LIN {X 0,Y 400.277,Z 579.545,A -85,B 0,C 180,E1 -11266.71,E2 -11266.71} C_VEL
LIN {X 0,Y 401.436,Z 567.994,A -85,B 0,C 180,E1 -11267.974,E2 -11267.974} C_VEL
LIN {X 0,Y 402.651,Z 555.178,A -85,B 0,C 180,E1 -11269.104,E2 -11269.104} C_VEL
LIN {X 0,Y 403.742,Z 541.629,A -85,B 0,C 180,E1 -11270.046,E2 -11270.046} C_VEL
LIN {X 0,Y 404.528,Z 528.73,A -85,B 0,C 180,E1 -11270.732,E2 -11270.732} C_VEL
LIN {X 0,Y 405.302,Z 514.967,A -85,B 0,C 180,E1 -11271.256,E2 -11271.256} C_VEL
LIN {X 0,Y 405.728,Z 500.889,A -85,B 0,C 180,E1 -11271.599,E2 -11271.599} C_VEL
LIN {X 0,Y 407.367,Z 401.658,A -85,B 0,C 180,E1 -11273.361,E2 -11273.361} C_VEL
LIN {X 0,Y 404.27,Z 384.321,A -85,B 0,C 180,E1 -11273.88,E2 -11273.88} C_VEL
LIN {X 0,Y 401.419,Z 370.358,A -85,B 0,C 180,E1 -11274.356,E2 -11274.356} C_VEL
LIN {X 0,Y 401.756,Z 366.638,A -85,B 0,C 180,E1 -11275.102,E2 -11275.102} C_VEL
LIN {X 0,Y 399.711,Z 355.979,A -85,B 0,C 180,E1 -11277.471,E2 -11277.471} C_VEL
LIN {X 0,Y 397.114,Z 344.644,A -85,B 0,C 180,E1 -11280.118,E2 -11280.118} C_VEL
LIN {X 0,Y 397.123,Z 344.645,A -85,B 0,C 180,E1 -11283.719,E2 -11283.719} C_VEL
LIN {X 0,Y 397.098,Z 344.645,A -85,B 0,C 180,E1 -11287.21,E2 -11287.21} C_VEL
LIN {X 0,Y 397.107,Z 344.641,A -85,B 0,C 180,E1 -11290.446,E2 -11290.446} C_VEL
LIN {X 0,Y 397.106,Z 344.644,A -85,B 0,C 180,E1 -11293.649,E2 -11293.649} C_VEL
LIN {X 0,Y 397.107,Z 344.643,A -85,B 0,C 180,E1 -11296.522,E2 -11296.522} C_VEL
LIN {X 0,Y 397.119,Z 344.642,A -85,B 0,C 180,E1 -11300.423,E2 -11300.423} C_VEL
LIN {X 0,Y 397.113,Z 344.646,A -85,B 0,C 180,E1 -11304.266,E2 -11304.266} C_VEL
LIN {X 0,Y 397.12,Z 344.644,A -85,B 0,C 180,E1 -11306.728,E2 -11306.728} C_VEL
LIN {X 0,Y 397.124,Z 344.649,A -85,B 0,C 180,E1 -11310.296,E2 -11310.296} C_VEL
LIN {X 0,Y 397.16,Z 344.763,A -85,B 0,C 180,E1 -11311.134,E2 -11311.134} C_VEL
LIN {X 0,Y 400.789,Z 356.95,A -85,B 0,C 180,E1 -11313.999,E2 -11313.999} C_VEL
LIN {X 0,Y 402.495,Z 364.53,A -85,B 0,C 180,E1 -11315.662,E2 -11315.662} C_VEL
LIN {X 0,Y 402.859,Z 369.281,A -85,B 0,C 180,E1 -11316.617,E2 -11316.617} C_VEL
LIN {X 0,Y 402.299,Z 381.598,A -85,B 0,C 180,E1 -11318.881,E2 -11318.881} C_VEL
LIN {X 0,Y 405.879,Z 396.627,A -85,B 0,C 180,E1 -11319.635,E2 -11319.635} C_VEL
LIN {X 0,Y 406.448,Z 400.682,A -85,B 0,C 180,E1 -11319.801,E2 -11319.801} C_VEL
LIN {X 0,Y 403.617,Z 480.645,A -85,B 0,C 180,E1 -11321.8,E2 -11321.8} C_VEL
LIN {X 0,Y 403.108,Z 495.536,A -85,B 0,C 180,E1 -11322.236,E2 -11322.236} C_VEL
LIN {X 0,Y 402.537,Z 508.176,A -85,B 0,C 180,E1 -11322.8,E2 -11322.8} C_VEL
LIN {X 0,Y 401.908,Z 519.55,A -85,B 0,C 180,E1 -11323.492,E2 -11323.492} C_VEL
LIN {X 0,Y 401.064,Z 531.353,A -85,B 0,C 180,E1 -11324.409,E2 -11324.409} C_VEL
LIN {X 0,Y 400.264,Z 541.681,A -85,B 0,C 180,E1 -11325.417,E2 -11325.417} C_VEL
LIN {X 0,Y 399.455,Z 550.912,A -85,B 0,C 180,E1 -11326.519,E2 -11326.519} C_VEL
LIN {X 0,Y 398.69,Z 559.636,A -85,B 0,C 180,E1 -11327.788,E2 -11327.788} C_VEL
LIN {X 0,Y 397.891,Z 568.178,A -85,B 0,C 180,E1 -11329.312,E2 -11329.312} C_VEL
LIN {X 0,Y 397.225,Z 574.98,A -85,B 0,C 180,E1 -11330.838,E2 -11330.838} C_VEL
LIN {X 0,Y 396.781,Z 580.383,A -85,B 0,C 180,E1 -11332.367,E2 -11332.367} C_VEL
LIN {X 0,Y 396.415,Z 584.568,A -85,B 0,C 180,E1 -11333.894,E2 -11333.894} C_VEL
LIN {X 0,Y 396.15,Z 586.768,A -85,B 0,C 180,E1 -11334.911,E2 -11334.911} C_VEL
LIN {X 0,Y 396.205,Z 588.437,A -85,B 0,C 180,E1 -11335.931,E2 -11335.931} C_VEL
LIN {X 0,Y 396.084,Z 589.693,A -85,B 0,C 180,E1 -11336.949,E2 -11336.949} C_VEL
LIN {X 0,Y 395.941,Z 590.539,A -85,B 0,C 180,E1 -11337.966,E2 -11337.966} C_VEL
LIN {X 0,Y 395.859,Z 590.913,A -85,B 0,C 180,E1 -11338.983,E2 -11338.983} C_VEL
LIN {X 0,Y 395.823,Z 590.865,A -85,B 0,C 180,E1 -11340,E2 -11340} C_VEL
LIN {X 0,Y 395.838,Z 590.407,A -85,B 0,C 180,E1 -11341.017,E2 -11341.017} C_VEL
LIN {X 0,Y 395.919,Z 589.489,A -85,B 0,C 180,E1 -11342.035,E2 -11342.035} C_VEL
LIN {X 0,Y 395.951,Z 588.135,A -85,B 0,C 180,E1 -11343.052,E2 -11343.052} C_VEL
LIN {X 0,Y 395.996,Z 585.27,A -85,B 0,C 180,E1 -11344.581,E2 -11344.581} C_VEL
LIN {X 0,Y 396.189,Z 581.317,A -85,B 0,C 180,E1 -11346.11,E2 -11346.11} C_VEL
LIN {X 0,Y 396.423,Z 576.171,A -85,B 0,C 180,E1 -11347.641,E2 -11347.641} C_VEL
LIN {X 0,Y 396.767,Z 569.656,A -85,B 0,C 180,E1 -11349.173,E2 -11349.173} C_VEL
LIN {X 0,Y 397.271,Z 561.487,A -85,B 0,C 180,E1 -11350.705,E2 -11350.705} C_VEL
LIN {X 0,Y 397.764,Z 553.153,A -85,B 0,C 180,E1 -11351.982,E2 -11351.982} C_VEL
LIN {X 0,Y 398.467,Z 542.953,A -85,B 0,C 180,E1 -11353.255,E2 -11353.255} C_VEL
LIN {X 0,Y 399.008,Z 532.049,A -85,B 0,C 180,E1 -11354.358,E2 -11354.358} C_VEL
LIN {X 0,Y 399.571,Z 520.38,A -85,B 0,C 180,E1 -11355.298,E2 -11355.298} C_VEL
LIN {X 0,Y 400.209,Z 506.876,A -85,B 0,C 180,E1 -11356.122,E2 -11356.122} C_VEL
LIN {X 0,Y 400.642,Z 493.868,A -85,B 0,C 180,E1 -11356.693,E2 -11356.693} C_VEL
LIN {X 0,Y 400.978,Z 479.075,A -85,B 0,C 180,E1 -11357.105,E2 -11357.105} C_VEL
LIN {X 0,Y 402.535,Z 397.502,A -85,B 0,C 180,E1 -11358.899,E2 -11358.899} C_VEL
LIN {X 0,Y 399.311,Z 377.922,A -85,B 0,C 180,E1 -11359.487,E2 -11359.487} C_VEL
LIN {X 0,Y 399.99,Z 360.43,A -85,B 0,C 180,E1 -11362.74,E2 -11362.74} C_VEL
LIN {X 0,Y 398.852,Z 353.072,A -85,B 0,C 180,E1 -11364.185,E2 -11364.185} C_VEL
LIN {X 0,Y 397.174,Z 344.638,A -85,B 0,C 180,E1 -11365.907,E2 -11365.907} C_VEL
LIN {X 0,Y 397.128,Z 344.643,A -85,B 0,C 180,E1 -11368.543,E2 -11368.543} C_VEL
LIN {X 0,Y 397.085,Z 344.649,A -85,B 0,C 180,E1 -11372.071,E2 -11372.071} C_VEL
LIN {X 0,Y 397.125,Z 344.642,A -85,B 0,C 180,E1 -11375.503,E2 -11375.503} C_VEL
LIN {X 0,Y 397.099,Z 344.643,A -85,B 0,C 180,E1 -11378.854,E2 -11378.854} C_VEL
LIN {X 0,Y 397.067,Z 344.65,A -85,B 0,C 180,E1 -11382.268,E2 -11382.268} C_VEL
LIN {X 0,Y 397.092,Z 344.646,A -85,B 0,C 180,E1 -11385.068,E2 -11385.068} C_VEL
LIN {X 0,Y 397.059,Z 344.651,A -85,B 0,C 180,E1 -11388.023,E2 -11388.023} C_VEL
LIN {X 0,Y 397.095,Z 344.648,A -85,B 0,C 180,E1 -11391.723,E2 -11391.723} C_VEL
LIN {X 0,Y 397.122,Z 344.641,A -85,B 0,C 180,E1 -11395.505,E2 -11395.505} C_VEL
LIN {X 0,Y 397.076,Z 344.649,A -85,B 0,C 180,E1 -11399.116,E2 -11399.116} C_VEL
LIN {X 0,Y 397.131,Z 344.765,A -85,B 0,C 180,E1 -11401.203,E2 -11401.203} C_VEL
LIN {X 0,Y 399.898,Z 357.338,A -85,B 0,C 180,E1 -11404.215,E2 -11404.215} C_VEL
LIN {X 0,Y 401.222,Z 363.882,A -85,B 0,C 180,E1 -11405.714,E2 -11405.714} C_VEL
LIN {X 0,Y 403.242,Z 371.317,A -85,B 0,C 180,E1 -11405.986,E2 -11405.986} C_VEL
LIN {X 0,Y 407.408,Z 391.656,A -85,B 0,C 180,E1 -11406.631,E2 -11406.631} C_VEL
LIN {X 0,Y 405.903,Z 489.536,A -85,B 0,C 180,E1 -11408.377,E2 -11408.377} C_VEL
LIN {X 0,Y 405.462,Z 505.277,A -85,B 0,C 180,E1 -11408.719,E2 -11408.719} C_VEL
LIN {X 0,Y 404.756,Z 519.212,A -85,B 0,C 180,E1 -11409.213,E2 -11409.213} C_VEL
LIN {X 0,Y 404.017,Z 532.788,A -85,B 0,C 180,E1 -11409.906,E2 -11409.906} C_VEL
LIN {X 0,Y 403.024,Z 545.847,A -85,B 0,C 180,E1 -11410.782,E2 -11410.782} C_VEL
LIN {X 0,Y 401.966,Z 557.736,A -85,B 0,C 180,E1 -11411.787,E2 -11411.787} C_VEL
LIN {X 0,Y 400.713,Z 569.777,A -85,B 0,C 180,E1 -11413.046,E2 -11413.046} C_VEL
LIN {X 0,Y 399.899,Z 577.879,A -85,B 0,C 180,E1 -11414.06,E2 -11414.06} C_VEL
LIN {X 0,Y 398.895,Z 580.792,A -85,B 0,C 180,E1 -11414.427,E2 -11414.427} C_VEL
LIN {X 0,Y 392.324,Z 589.579,A -85,B 0,C 180,E1 -11415.574,E2 -11415.574} C_VEL
LIN {X 0,Y 391.485,Z 592.107,A -85,B 0,C 180,E1 -11416.004,E2 -11416.004} C_VEL
LIN {X 0,Y 390.581,Z 600.976,A -85,B 0,C 180,E1 -11417.793,E2 -11417.793} C_VEL
LIN {X 0,Y 389.828,Z 608.252,A -85,B 0,C 180,E1 -11419.612,E2 -11419.612} C_VEL
LIN {X 0,Y 389.212,Z 614.788,A -85,B 0,C 180,E1 -11421.693,E2 -11421.693} C_VEL
LIN {X 0,Y 388.924,Z 619.682,A -85,B 0,C 180,E1 -11423.774,E2 -11423.774} C_VEL
LIN {X 0,Y 388.718,Z 623.093,A -85,B 0,C 180,E1 -11425.851,E2 -11425.851} C_VEL
LIN {X 0,Y 388.66,Z 625.122,A -85,B 0,C 180,E1 -11427.926,E2 -11427.926} C_VEL
LIN {X 0,Y 388.672,Z 625.82,A -85,B 0,C 180,E1 -11429.998,E2 -11429.998} C_VEL
LIN {X 0,Y 388.659,Z 625.196,A -85,B 0,C 180,E1 -11432.071,E2 -11432.071} C_VEL
LIN {X 0,Y 388.716,Z 623.237,A -85,B 0,C 180,E1 -11434.146,E2 -11434.146} C_VEL
LIN {X 0,Y 388.873,Z 619.891,A -85,B 0,C 180,E1 -11436.224,E2 -11436.224} C_VEL
LIN {X 0,Y 389.207,Z 615.06,A -85,B 0,C 180,E1 -11438.304,E2 -11438.304} C_VEL
LIN {X 0,Y 389.799,Z 608.599,A -85,B 0,C 180,E1 -11440.385,E2 -11440.385} C_VEL
LIN {X 0,Y 390.544,Z 601.405,A -85,B 0,C 180,E1 -11442.205,E2 -11442.205} C_VEL
LIN {X 0,Y 391.402,Z 592.717,A -85,B 0,C 180,E1 -11443.987,E2 -11443.987} C_VEL
LIN {X 0,Y 392.456,Z 583.155,A -85,B 0,C 180,E1 -11445.58,E2 -11445.58} C_VEL
LIN {X 0,Y 393.642,Z 572.796,A -85,B 0,C 180,E1 -11446.997,E2 -11446.997} C_VEL
LIN {X 0,Y 394.857,Z 561.37,A -85,B 0,C 180,E1 -11448.281,E2 -11448.281} C_VEL
LIN {X 0,Y 396.091,Z 548.705,A -85,B 0,C 180,E1 -11449.43,E2 -11449.43} C_VEL
LIN {X 0,Y 397.149,Z 535.171,A -85,B 0,C 180,E1 -11450.402,E2 -11450.402} C_VEL
LIN {X 0,Y 398.085,Z 521.413,A -85,B 0,C 180,E1 -11451.148,E2 -11451.148} C_VEL
LIN {X 0,Y 398.801,Z 507.58,A -85,B 0,C 180,E1 -11451.685,E2 -11451.685} C_VEL
LIN {X 0,Y 399.296,Z 493.25,A -85,B 0,C 180,E1 -11452.03,E2 -11452.03} C_VEL
LIN {X 0,Y 400.989,Z 393.489,A -85,B 0,C 180,E1 -11453.832,E2 -11453.832} C_VEL
LIN {X 0,Y 396.082,Z 369.523,A -85,B 0,C 180,E1 -11454.614,E2 -11454.614} C_VEL
LIN {X 0,Y 394.027,Z 363.86,A -85,B 0,C 180,E1 -11454.87,E2 -11454.87} C_VEL
LIN {X 0,Y 391.431,Z 351.504,A -85,B 0,C 180,E1 -11457.826,E2 -11457.826} C_VEL
LIN {X 0,Y 390.083,Z 345.525,A -85,B 0,C 180,E1 -11459.327,E2 -11459.327} C_VEL
LIN {X 0,Y 390.036,Z 345.531,A -85,B 0,C 180,E1 -11462.72,E2 -11462.72} C_VEL
LIN {X 0,Y 390.048,Z 345.525,A -85,B 0,C 180,E1 -11465.823,E2 -11465.823} C_VEL
LIN {X 0,Y 390.029,Z 345.527,A -85,B 0,C 180,E1 -11469.211,E2 -11469.211} C_VEL
LIN {X 0,Y 390.021,Z 345.527,A -85,B 0,C 180,E1 -11472.37,E2 -11472.37} C_VEL
LIN {X 0,Y 390.033,Z 345.525,A -85,B 0,C 180,E1 -11475.352,E2 -11475.352} C_VEL
LIN {X 0,Y 390.005,Z 345.528,A -85,B 0,C 180,E1 -11478.183,E2 -11478.183} C_VEL
LIN {X 0,Y 390.047,Z 345.519,A -85,B 0,C 180,E1 -11480.902,E2 -11480.902} C_VEL
LIN {X 0,Y 390.07,Z 345.524,A -85,B 0,C 180,E1 -11484.791,E2 -11484.791} C_VEL
LIN {X 0,Y 390.009,Z 345.52,A -85,B 0,C 180,E1 -11488.494,E2 -11488.494} C_VEL
LIN {X 0,Y 390.002,Z 345.524,A -85,B 0,C 180,E1 -11492.002,E2 -11492.002} C_VEL
LIN {X 0,Y 390.029,Z 345.522,A -85,B 0,C 180,E1 -11495.516,E2 -11495.516} C_VEL
LIN {X 0,Y 390.041,Z 345.517,A -85,B 0,C 180,E1 -11498.877,E2 -11498.877} C_VEL
LIN {X 0,Y 390.097,Z 345.504,A -85,B 0,C 180,E1 -11502.165,E2 -11502.165} C_VEL
LIN {X 0,Y 390.126,Z 345.511,A -85,B 0,C 180,E1 -11505.392,E2 -11505.392} C_VEL
LIN {X 0,Y 390.13,Z 345.515,A -85,B 0,C 180,E1 -11508.571,E2 -11508.571} C_VEL
LIN {X 0,Y 390.241,Z 345.495,A -85,B 0,C 180,E1 -11512.086,E2 -11512.086} C_VEL
LIN {X 0,Y 390.184,Z 345.502,A -85,B 0,C 180,E1 -11514.833,E2 -11514.833} C_VEL
LIN {X 0,Y 390.395,Z 345.479,A -85,B 0,C 180,E1 -11517.937,E2 -11517.937} C_VEL
LIN {X 0,Y 390.392,Z 345.48,A -85,B 0,C 180,E1 -11522.063,E2 -11522.063} C_VEL
LIN {X 0,Y 390.269,Z 345.496,A -85,B 0,C 180,E1 -11526.203,E2 -11526.203} C_VEL
LIN {X 0,Y 390.17,Z 345.504,A -85,B 0,C 180,E1 -11529.33,E2 -11529.33} C_VEL
LIN {X 0,Y 390.18,Z 345.502,A -85,B 0,C 180,E1 -11533.439,E2 -11533.439} C_VEL
LIN {X 0,Y 390.115,Z 345.51,A -85,B 0,C 180,E1 -11537.299,E2 -11537.299} C_VEL
LIN {X 0,Y 390.074,Z 345.514,A -85,B 0,C 180,E1 -11540.471,E2 -11540.471} C_VEL
LIN {X 0,Y 390.043,Z 345.513,A -85,B 0,C 180,E1 -11543.354,E2 -11543.354} C_VEL
LIN {X 0,Y 390.018,Z 345.524,A -85,B 0,C 180,E1 -11546.775,E2 -11546.775} C_VEL
LIN {X 0,Y 390.023,Z 345.52,A -85,B 0,C 180,E1 -11550.301,E2 -11550.301} C_VEL
LIN {X 0,Y 390.056,Z 345.521,A -85,B 0,C 180,E1 -11554.026,E2 -11554.026} C_VEL
LIN {X 0,Y 390.023,Z 345.527,A -85,B 0,C 180,E1 -11557.782,E2 -11557.782} C_VEL
LIN {X 0,Y 390.004,Z 345.527,A -85,B 0,C 180,E1 -11560.816,E2 -11560.816} C_VEL
LIN {X 0,Y 390.032,Z 345.525,A -85,B 0,C 180,E1 -11563.886,E2 -11563.886} C_VEL
LIN {X 0,Y 390.036,Z 345.527,A -85,B 0,C 180,E1 -11566.789,E2 -11566.789} C_VEL
LIN {X 0,Y 390,Z 345.531,A -85,B 0,C 180,E1 -11569.556,E2 -11569.556} C_VEL
LIN {X 0,Y 390.027,Z 345.53,A -85,B 0,C 180,E1 -11572.452,E2 -11572.452} C_VEL
LIN {X 0,Y 390.054,Z 345.526,A -85,B 0,C 180,E1 -11576.046,E2 -11576.046} C_VEL
LIN {X 0,Y 390.071,Z 345.654,A -85,B 0,C 180,E1 -11579.518,E2 -11579.518} C_VEL
LIN {X 0,Y 393.033,Z 358.498,A -85,B 0,C 180,E1 -11582.566,E2 -11582.566} C_VEL
LIN {X 0,Y 394.863,Z 367.974,A -85,B 0,C 180,E1 -11584.714,E2 -11584.714} C_VEL
LIN {X 0,Y 394.674,Z 370.357,A -85,B 0,C 180,E1 -11585.203,E2 -11585.203} C_VEL
LIN {X 0,Y 400.422,Z 399.362,A -85,B 0,C 180,E1 -11586.156,E2 -11586.156} C_VEL
LIN {X 0,Y 400.86,Z 403.279,A -85,B 0,C 180,E1 -11586.259,E2 -11586.259} C_VEL
LIN {X 0,Y 399.023,Z 507.416,A -85,B 0,C 180,E1 -11588.158,E2 -11588.158} C_VEL
LIN {X 0,Y 398.362,Z 521.51,A -85,B 0,C 180,E1 -11588.596,E2 -11588.596} C_VEL
LIN {X 0,Y 397.48,Z 535.196,A -85,B 0,C 180,E1 -11589.225,E2 -11589.225} C_VEL
LIN {X 0,Y 396.474,Z 548.971,A -85,B 0,C 180,E1 -11590.087,E2 -11590.087} C_VEL
LIN {X 0,Y 395.362,Z 561.288,A -85,B 0,C 180,E1 -11591.072,E2 -11591.072} C_VEL
LIN {X 0,Y 394.149,Z 572.919,A -85,B 0,C 180,E1 -11592.222,E2 -11592.222} C_VEL
LIN {X 0,Y 393.09,Z 582.602,A -85,B 0,C 180,E1 -11593.379,E2 -11593.379} C_VEL
LIN {X 0,Y 391.871,Z 593.332,A -85,B 0,C 180,E1 -11594.929,E2 -11594.929} C_VEL
LIN {X 0,Y 390.958,Z 602.191,A -85,B 0,C 180,E1 -11596.487,E2 -11596.487} C_VEL
LIN {X 0,Y 390.267,Z 609.564,A -85,B 0,C 180,E1 -11598.05,E2 -11598.05} C_VEL
LIN {X 0,Y 389.589,Z 615.708,A -85,B 0,C 180,E1 -11599.609,E2 -11599.609} C_VEL
LIN {X 0,Y 389.09,Z 622.234,A -85,B 0,C 180,E1 -11601.693,E2 -11601.693} C_VEL
LIN {X 0,Y 388.802,Z 627.209,A -85,B 0,C 180,E1 -11603.817,E2 -11603.817} C_VEL
LIN {X 0,Y 388.681,Z 630.52,A -85,B 0,C 180,E1 -11605.854,E2 -11605.854} C_VEL
LIN {X 0,Y 388.613,Z 632.525,A -85,B 0,C 180,E1 -11607.929,E2 -11607.929} C_VEL
LIN {X 0,Y 388.671,Z 633.187,A -85,B 0,C 180,E1 -11610.002,E2 -11610.002} C_VEL
LIN {X 0,Y 388.614,Z 632.516,A -85,B 0,C 180,E1 -11612.074,E2 -11612.074} C_VEL
LIN {X 0,Y 388.681,Z 630.502,A -85,B 0,C 180,E1 -11614.149,E2 -11614.149} C_VEL
LIN {X 0,Y 388.835,Z 627.099,A -85,B 0,C 180,E1 -11616.227,E2 -11616.227} C_VEL
LIN {X 0,Y 389.093,Z 622.207,A -85,B 0,C 180,E1 -11618.31,E2 -11618.31} C_VEL
LIN {X 0,Y 389.593,Z 615.67,A -85,B 0,C 180,E1 -11620.394,E2 -11620.394} C_VEL
LIN {X 0,Y 390.367,Z 608.398,A -85,B 0,C 180,E1 -11622.214,E2 -11622.214} C_VEL
LIN {X 0,Y 391.12,Z 600.545,A -85,B 0,C 180,E1 -11623.82,E2 -11623.82} C_VEL
LIN {X 0,Y 392.048,Z 591.631,A -85,B 0,C 180,E1 -11625.334,E2 -11625.334} C_VEL
LIN {X 0,Y 393.342,Z 580.542,A -85,B 0,C 180,E1 -11626.88,E2 -11626.88} C_VEL
LIN {X 0,Y 394.533,Z 569.216,A -85,B 0,C 180,E1 -11628.165,E2 -11628.165} C_VEL
LIN {X 0,Y 395.779,Z 556.688,A -85,B 0,C 180,E1 -11629.315,E2 -11629.315} C_VEL
LIN {X 0,Y 396.912,Z 543.713,A -85,B 0,C 180,E1 -11630.259,E2 -11630.259} C_VEL
LIN {X 0,Y 397.796,Z 529.957,A -85,B 0,C 180,E1 -11631.032,E2 -11631.032} C_VEL
LIN {X 0,Y 398.651,Z 515.806,A -85,B 0,C 180,E1 -11631.595,E2 -11631.595} C_VEL
LIN {X 0,Y 399.113,Z 502.36,A -85,B 0,C 180,E1 -11631.942,E2 -11631.942} C_VEL
LIN {X 0,Y 400.848,Z 404.818,A -85,B 0,C 180,E1 -11633.702,E2 -11633.702} C_VEL
LIN {X 0,Y 400.532,Z 399.888,A -85,B 0,C 180,E1 -11633.817,E2 -11633.817} C_VEL
LIN {X 0,Y 394.671,Z 370.347,A -85,B 0,C 180,E1 -11634.788,E2 -11634.788} C_VEL
LIN {X 0,Y 394.677,Z 366.564,A -85,B 0,C 180,E1 -11635.584,E2 -11635.584} C_VEL
LIN {X 0,Y 391.99,Z 353.714,A -85,B 0,C 180,E1 -11638.535,E2 -11638.535} C_VEL
LIN {X 0,Y 390.058,Z 345.525,A -85,B 0,C 180,E1 -11640.524,E2 -11640.524} C_VEL
LIN {X 0,Y 390.073,Z 345.521,A -85,B 0,C 180,E1 -11644.026,E2 -11644.026} C_VEL
LIN {X 0,Y 390.047,Z 345.524,A -85,B 0,C 180,E1 -11647.551,E2 -11647.551} C_VEL
LIN {X 0,Y 390.061,Z 345.52,A -85,B 0,C 180,E1 -11650.822,E2 -11650.822} C_VEL
LIN {X 0,Y 390.06,Z 345.522,A -85,B 0,C 180,E1 -11653.887,E2 -11653.887} C_VEL
LIN {X 0,Y 390.062,Z 345.522,A -85,B 0,C 180,E1 -11656.79,E2 -11656.79} C_VEL
LIN {X 0,Y 390.062,Z 345.521,A -85,B 0,C 180,E1 -11659.561,E2 -11659.561} C_VEL
LIN {X 0,Y 390.048,Z 345.524,A -85,B 0,C 180,E1 -11662.45,E2 -11662.45} C_VEL
LIN {X 0,Y 390.074,Z 345.524,A -85,B 0,C 180,E1 -11666.046,E2 -11666.046} C_VEL
LIN {X 0,Y 390.05,Z 345.53,A -85,B 0,C 180,E1 -11669.87,E2 -11669.87} C_VEL
LIN {X 0,Y 390.08,Z 345.542,A -85,B 0,C 180,E1 -11670.3,E2 -11670.3} C_VEL
LIN {X 0,Y 393.751,Z 357.145,A -85,B 0,C 180,E1 -11673.184,E2 -11673.184} C_VEL
LIN {X 0,Y 395.963,Z 366.556,A -85,B 0,C 180,E1 -11675.32,E2 -11675.32} C_VEL
LIN {X 0,Y 396.421,Z 370.831,A -85,B 0,C 180,E1 -11676.214,E2 -11676.214} C_VEL
LIN {X 0,Y 395.855,Z 382.001,A -85,B 0,C 180,E1 -11678.311,E2 -11678.311} C_VEL
LIN {X 0,Y 399.364,Z 396.308,A -85,B 0,C 180,E1 -11679.08,E2 -11679.08} C_VEL
LIN {X 0,Y 400.252,Z 401.562,A -85,B 0,C 180,E1 -11679.32,E2 -11679.32} C_VEL
LIN {X 0,Y 397.189,Z 480.415,A -85,B 0,C 180,E1 -11681.361,E2 -11681.361} C_VEL
LIN {X 0,Y 396.65,Z 495.328,A -85,B 0,C 180,E1 -11681.803,E2 -11681.803} C_VEL
LIN {X 0,Y 396.046,Z 508.049,A -85,B 0,C 180,E1 -11682.375,E2 -11682.375} C_VEL
LIN {X 0,Y 395.342,Z 519.518,A -85,B 0,C 180,E1 -11683.076,E2 -11683.076} C_VEL
LIN {X 0,Y 394.463,Z 531.491,A -85,B 0,C 180,E1 -11684.022,E2 -11684.022} C_VEL
LIN {X 0,Y 393.51,Z 542.814,A -85,B 0,C 180,E1 -11685.154,E2 -11685.154} C_VEL
LIN {X 0,Y 392.392,Z 553.857,A -85,B 0,C 180,E1 -11686.536,E2 -11686.536} C_VEL
LIN {X 0,Y 391.644,Z 562.12,A -85,B 0,C 180,E1 -11687.828,E2 -11687.828} C_VEL
LIN {X 0,Y 390.865,Z 570.195,A -85,B 0,C 180,E1 -11689.38,E2 -11689.38} C_VEL
LIN {X 0,Y 390.263,Z 575.699,A -85,B 0,C 180,E1 -11690.673,E2 -11690.673} C_VEL
LIN {X 0,Y 389.78,Z 581.03,A -85,B 0,C 180,E1 -11692.228,E2 -11692.228} C_VEL
LIN {X 0,Y 389.387,Z 585.154,A -85,B 0,C 180,E1 -11693.783,E2 -11693.783} C_VEL
LIN {X 0,Y 389.094,Z 587.299,A -85,B 0,C 180,E1 -11694.818,E2 -11694.818} C_VEL
LIN {X 0,Y 389.135,Z 588.926,A -85,B 0,C 180,E1 -11695.857,E2 -11695.857} C_VEL
LIN {X 0,Y 389.03,Z 590.148,A -85,B 0,C 180,E1 -11696.893,E2 -11696.893} C_VEL
LIN {X 0,Y 388.878,Z 590.946,A -85,B 0,C 180,E1 -11697.929,E2 -11697.929} C_VEL
LIN {X 0,Y 388.788,Z 591.276,A -85,B 0,C 180,E1 -11698.964,E2 -11698.964} C_VEL
LIN {X 0,Y 388.75,Z 591.192,A -85,B 0,C 180,E1 -11700,E2 -11700} C_VEL
LIN {X 0,Y 388.768,Z 590.69,A -85,B 0,C 180,E1 -11701.036,E2 -11701.036} C_VEL
LIN {X 0,Y 388.835,Z 589.714,A -85,B 0,C 180,E1 -11702.072,E2 -11702.072} C_VEL
LIN {X 0,Y 388.854,Z 588.322,A -85,B 0,C 180,E1 -11703.108,E2 -11703.108} C_VEL
LIN {X 0,Y 388.931,Z 585.378,A -85,B 0,C 180,E1 -11704.664,E2 -11704.664} C_VEL
LIN {X 0,Y 389.118,Z 581.341,A -85,B 0,C 180,E1 -11706.221,E2 -11706.221} C_VEL
LIN {X 0,Y 389.358,Z 576.096,A -85,B 0,C 180,E1 -11707.781,E2 -11707.781} C_VEL
LIN {X 0,Y 389.736,Z 569.434,A -85,B 0,C 180,E1 -11709.34,E2 -11709.34} C_VEL
LIN {X 0,Y 390.235,Z 561.133,A -85,B 0,C 180,E1 -11710.9,E2 -11710.9} C_VEL
LIN {X 0,Y 390.789,Z 552.648,A -85,B 0,C 180,E1 -11712.199,E2 -11712.199} C_VEL
LIN {X 0,Y 391.452,Z 542.201,A -85,B 0,C 180,E1 -11713.497,E2 -11713.497} C_VEL
LIN {X 0,Y 392.089,Z 530.527,A -85,B 0,C 180,E1 -11714.666,E2 -11714.666} C_VEL
LIN {X 0,Y 392.662,Z 518.966,A -85,B 0,C 180,E1 -11715.574,E2 -11715.574} C_VEL
LIN {X 0,Y 393.289,Z 506.215,A -85,B 0,C 180,E1 -11716.347,E2 -11716.347} C_VEL
LIN {X 0,Y 393.719,Z 492.724,A -85,B 0,C 180,E1 -11716.929,E2 -11716.929} C_VEL
LIN {X 0,Y 394.04,Z 478.712,A -85,B 0,C 180,E1 -11717.316,E2 -11717.316} C_VEL
LIN {X 0,Y 395.663,Z 398.492,A -85,B 0,C 180,E1 -11719.133,E2 -11719.133} C_VEL
LIN {X 0,Y 392.379,Z 378.146,A -85,B 0,C 180,E1 -11719.759,E2 -11719.759} C_VEL
LIN {X 0,Y 393.039,Z 361.462,A -85,B 0,C 180,E1 -11722.887,E2 -11722.887} C_VEL
LIN {X 0,Y 391.522,Z 352.494,A -85,B 0,C 180,E1 -11724.667,E2 -11724.667} C_VEL
LIN {X 0,Y 390.141,Z 345.515,A -85,B 0,C 180,E1 -11726.084,E2 -11726.084} C_VEL
LIN {X 0,Y 390.064,Z 345.52,A -85,B 0,C 180,E1 -11729.109,E2 -11729.109} C_VEL
LIN {X 0,Y 390.049,Z 345.522,A -85,B 0,C 180,E1 -11732.721,E2 -11732.721} C_VEL
LIN {X 0,Y 390.061,Z 345.524,A -85,B 0,C 180,E1 -11735.825,E2 -11735.825} C_VEL
LIN {X 0,Y 390.043,Z 345.522,A -85,B 0,C 180,E1 -11739.212,E2 -11739.212} C_VEL
LIN {X 0,Y 390.042,Z 345.524,A -85,B 0,C 180,E1 -11742.373,E2 -11742.373} C_VEL
LIN {X 0,Y 390.049,Z 345.525,A -85,B 0,C 180,E1 -11745.353,E2 -11745.353} C_VEL
LIN {X 0,Y 390.022,Z 345.527,A -85,B 0,C 180,E1 -11748.184,E2 -11748.184} C_VEL
LIN {X 0,Y 390.062,Z 345.522,A -85,B 0,C 180,E1 -11750.903,E2 -11750.903} C_VEL
LIN {X 0,Y 390.074,Z 345.519,A -85,B 0,C 180,E1 -11754.791,E2 -11754.791} C_VEL
LIN {X 0,Y 390.022,Z 345.529,A -85,B 0,C 180,E1 -11758.494,E2 -11758.494} C_VEL
LIN {X 0,Y 390.091,Z 345.629,A -85,B 0,C 180,E1 -11760.818,E2 -11760.818} C_VEL
LIN {X 0,Y 393.019,Z 358.821,A -85,B 0,C 180,E1 -11764.045,E2 -11764.045} C_VEL
LIN {X 0,Y 394.088,Z 364.135,A -85,B 0,C 180,E1 -11765.248,E2 -11765.248} C_VEL
LIN {X 0,Y 396.357,Z 370.651,A -85,B 0,C 180,E1 -11765.527,E2 -11765.527} C_VEL
LIN {X 0,Y 400.941,Z 393.402,A -85,B 0,C 180,E1 -11766.263,E2 -11766.263} C_VEL
LIN {X 0,Y 399.139,Z 497.863,A -85,B 0,C 180,E1 -11768.162,E2 -11768.162} C_VEL
LIN {X 0,Y 398.592,Z 512.141,A -85,B 0,C 180,E1 -11768.572,E2 -11768.572} C_VEL
LIN {X 0,Y 397.864,Z 524.655,A -85,B 0,C 180,E1 -11769.107,E2 -11769.107} C_VEL
LIN {X 0,Y 396.904,Z 538.586,A -85,B 0,C 180,E1 -11769.917,E2 -11769.917} C_VEL
LIN {X 0,Y 395.874,Z 550.66,A -85,B 0,C 180,E1 -11770.825,E2 -11770.825} C_VEL
LIN {X 0,Y 394.715,Z 562.953,A -85,B 0,C 180,E1 -11771.978,E2 -11771.978} C_VEL
LIN {X 0,Y 393.576,Z 573.051,A -85,B 0,C 180,E1 -11773.13,E2 -11773.13} C_VEL
LIN {X 0,Y 392.489,Z 582.475,A -85,B 0,C 180,E1 -11774.418,E2 -11774.418} C_VEL
LIN {X 0,Y 391.485,Z 592.107,A -85,B 0,C 180,E1 -11776.004,E2 -11776.004} C_VEL
LIN {X 0,Y 390.592,Z 595.757,A -85,B 0,C 180,E1 -11776.675,E2 -11776.675} C_VEL
LIN {X 0,Y 387.181,Z 601.366,A -85,B 0,C 180,E1 -11777.769,E2 -11777.769} C_VEL
LIN {X 0,Y 383.695,Z 606.461,A -85,B 0,C 180,E1 -11778.928,E2 -11778.928} C_VEL
LIN {X 0,Y 382.704,Z 609.251,A -85,B 0,C 180,E1 -11779.692,E2 -11779.692} C_VEL
LIN {X 0,Y 382.159,Z 614.857,A -85,B 0,C 180,E1 -11781.538,E2 -11781.538} C_VEL
LIN {X 0,Y 381.85,Z 619.751,A -85,B 0,C 180,E1 -11783.658,E2 -11783.658} C_VEL
LIN {X 0,Y 381.647,Z 623.16,A -85,B 0,C 180,E1 -11785.774,E2 -11785.774} C_VEL
LIN {X 0,Y 381.558,Z 625.189,A -85,B 0,C 180,E1 -11787.887,E2 -11787.887} C_VEL
LIN {X 0,Y 381.572,Z 625.887,A -85,B 0,C 180,E1 -11789.998,E2 -11789.998} C_VEL
LIN {X 0,Y 381.557,Z 625.263,A -85,B 0,C 180,E1 -11792.11,E2 -11792.11} C_VEL
LIN {X 0,Y 381.645,Z 623.303,A -85,B 0,C 180,E1 -11794.223,E2 -11794.223} C_VEL
LIN {X 0,Y 381.807,Z 619.957,A -85,B 0,C 180,E1 -11796.339,E2 -11796.339} C_VEL
LIN {X 0,Y 382.153,Z 615.126,A -85,B 0,C 180,E1 -11798.459,E2 -11798.459} C_VEL
LIN {X 0,Y 382.773,Z 608.665,A -85,B 0,C 180,E1 -11800.578,E2 -11800.578} C_VEL
LIN {X 0,Y 383.58,Z 601.471,A -85,B 0,C 180,E1 -11802.43,E2 -11802.43} C_VEL
LIN {X 0,Y 384.416,Z 593.319,A -85,B 0,C 180,E1 -11804.139,E2 -11804.139} C_VEL
LIN {X 0,Y 385.399,Z 584.875,A -85,B 0,C 180,E1 -11805.601,E2 -11805.601} C_VEL
LIN {X 0,Y 386.712,Z 573.904,A -85,B 0,C 180,E1 -11807.175,E2 -11807.175} C_VEL
LIN {X 0,Y 387.982,Z 562.72,A -85,B 0,C 180,E1 -11808.48,E2 -11808.48} C_VEL
LIN {X 0,Y 389.255,Z 550.346,A -85,B 0,C 180,E1 -11809.648,E2 -11809.648} C_VEL
LIN {X 0,Y 390.306,Z 537.716,A -85,B 0,C 180,E1 -11810.603,E2 -11810.603} C_VEL
LIN {X 0,Y 391.306,Z 524.07,A -85,B 0,C 180,E1 -11811.395,E2 -11811.395} C_VEL
LIN {X 0,Y 392.109,Z 509.468,A -85,B 0,C 180,E1 -11812.005,E2 -11812.005} C_VEL
LIN {X 0,Y 392.704,Z 494.938,A -85,B 0,C 180,E1 -11812.385,E2 -11812.385} C_VEL
LIN {X 0,Y 394.491,Z 394.763,A -85,B 0,C 180,E1 -11814.226,E2 -11814.226} C_VEL
LIN {X 0,Y 390.195,Z 373.29,A -85,B 0,C 180,E1 -11814.937,E2 -11814.937} C_VEL
LIN {X 0,Y 388.077,Z 367.022,A -85,B 0,C 180,E1 -11815.208,E2 -11815.208} C_VEL
LIN {X 0,Y 386.824,Z 363.961,A -85,B 0,C 180,E1 -11815.358,E2 -11815.358} C_VEL
LIN {X 0,Y 384.222,Z 351.572,A -85,B 0,C 180,E1 -11818.395,E2 -11818.395} C_VEL
LIN {X 0,Y 383.015,Z 346.405,A -85,B 0,C 180,E1 -11819.755,E2 -11819.755} C_VEL
LIN {X 0,Y 382.997,Z 346.406,A -85,B 0,C 180,E1 -11823.399,E2 -11823.399} C_VEL
LIN {X 0,Y 383.024,Z 346.4,A -85,B 0,C 180,E1 -11826.162,E2 -11826.162} C_VEL
LIN {X 0,Y 382.966,Z 346.405,A -85,B 0,C 180,E1 -11829.961,E2 -11829.961} C_VEL
LIN {X 0,Y 382.997,Z 346.402,A -85,B 0,C 180,E1 -11832.777,E2 -11832.777} C_VEL
LIN {X 0,Y 382.985,Z 346.401,A -85,B 0,C 180,E1 -11835.787,E2 -11835.787} C_VEL
LIN {X 0,Y 382.951,Z 346.408,A -85,B 0,C 180,E1 -11838.799,E2 -11838.799} C_VEL
LIN {X 0,Y 382.982,Z 346.393,A -85,B 0,C 180,E1 -11842.096,E2 -11842.096} C_VEL
LIN {X 0,Y 383.005,Z 346.398,A -85,B 0,C 180,E1 -11845.331,E2 -11845.331} C_VEL
LIN {X 0,Y 382.969,Z 346.405,A -85,B 0,C 180,E1 -11849.08,E2 -11849.08} C_VEL
LIN {X 0,Y 382.957,Z 346.394,A -85,B 0,C 180,E1 -11852.69,E2 -11852.69} C_VEL
LIN {X 0,Y 382.996,Z 346.399,A -85,B 0,C 180,E1 -11856.19,E2 -11856.19} C_VEL
LIN {X 0,Y 383.042,Z 346.383,A -85,B 0,C 180,E1 -11859.598,E2 -11859.598} C_VEL
LIN {X 0,Y 383.08,Z 346.387,A -85,B 0,C 180,E1 -11862.93,E2 -11862.93} C_VEL
LIN {X 0,Y 383.112,Z 346.386,A -85,B 0,C 180,E1 -11866.463,E2 -11866.463} C_VEL
LIN {X 0,Y 383.127,Z 346.384,A -85,B 0,C 180,E1 -11870.497,E2 -11870.497} C_VEL
LIN {X 0,Y 383.214,Z 346.372,A -85,B 0,C 180,E1 -11873.682,E2 -11873.682} C_VEL
LIN {X 0,Y 383.361,Z 346.355,A -85,B 0,C 180,E1 -11877.899,E2 -11877.899} C_VEL
LIN {X 0,Y 383.358,Z 346.356,A -85,B 0,C 180,E1 -11882.101,E2 -11882.101} C_VEL
LIN {X 0,Y 383.225,Z 346.375,A -85,B 0,C 180,E1 -11886.317,E2 -11886.317} C_VEL
LIN {X 0,Y 383.121,Z 346.382,A -85,B 0,C 180,E1 -11889.503,E2 -11889.503} C_VEL
LIN {X 0,Y 383.111,Z 346.382,A -85,B 0,C 180,E1 -11893.536,E2 -11893.536} C_VEL
LIN {X 0,Y 383.08,Z 346.387,A -85,B 0,C 180,E1 -11897.07,E2 -11897.07} C_VEL
LIN {X 0,Y 383.015,Z 346.391,A -85,B 0,C 180,E1 -11900.647,E2 -11900.647} C_VEL
LIN {X 0,Y 382.994,Z 346.392,A -85,B 0,C 180,E1 -11903.81,E2 -11903.81} C_VEL
LIN {X 0,Y 382.957,Z 346.401,A -85,B 0,C 180,E1 -11907.31,E2 -11907.31} C_VEL
LIN {X 0,Y 382.968,Z 346.405,A -85,B 0,C 180,E1 -11910.92,E2 -11910.92} C_VEL
LIN {X 0,Y 382.998,Z 346.402,A -85,B 0,C 180,E1 -11914.67,E2 -11914.67} C_VEL
LIN {X 0,Y 382.979,Z 346.405,A -85,B 0,C 180,E1 -11917.903,E2 -11917.903} C_VEL
LIN {X 0,Y 382.948,Z 346.405,A -85,B 0,C 180,E1 -11921.352,E2 -11921.352} C_VEL
LIN {X 0,Y 382.978,Z 346.408,A -85,B 0,C 180,E1 -11924.303,E2 -11924.303} C_VEL
LIN {X 0,Y 382.972,Z 346.405,A -85,B 0,C 180,E1 -11927.238,E2 -11927.238} C_VEL
LIN {X 0,Y 382.974,Z 346.409,A -85,B 0,C 180,E1 -11930.421,E2 -11930.421} C_VEL
LIN {X 0,Y 383.004,Z 346.405,A -85,B 0,C 180,E1 -11934.045,E2 -11934.045} C_VEL
LIN {X 0,Y 382.977,Z 346.406,A -85,B 0,C 180,E1 -11937.58,E2 -11937.58} C_VEL
LIN {X 0,Y 383.007,Z 346.428,A -85,B 0,C 180,E1 -11939.086,E2 -11939.086} C_VEL
LIN {X 0,Y 386.126,Z 359.868,A -85,B 0,C 180,E1 -11942.349,E2 -11942.349} C_VEL
LIN {X 0,Y 387.969,Z 369.226,A -85,B 0,C 180,E1 -11944.516,E2 -11944.516} C_VEL
LIN {X 0,Y 387.918,Z 370.33,A -85,B 0,C 180,E1 -11944.75,E2 -11944.75} C_VEL
LIN {X 0,Y 393.841,Z 399.763,A -85,B 0,C 180,E1 -11945.741,E2 -11945.741} C_VEL
LIN {X 0,Y 394.377,Z 403.386,A -85,B 0,C 180,E1 -11945.847,E2 -11945.847} C_VEL
LIN {X 0,Y 392.453,Z 507.364,A -85,B 0,C 180,E1 -11947.773,E2 -11947.773} C_VEL
LIN {X 0,Y 391.771,Z 521.451,A -85,B 0,C 180,E1 -11948.218,E2 -11948.218} C_VEL
LIN {X 0,Y 390.866,Z 535.135,A -85,B 0,C 180,E1 -11948.857,E2 -11948.857} C_VEL
LIN {X 0,Y 389.831,Z 548.385,A -85,B 0,C 180,E1 -11949.692,E2 -11949.692} C_VEL
LIN {X 0,Y 388.645,Z 561.225,A -85,B 0,C 180,E1 -11950.732,E2 -11950.732} C_VEL
LIN {X 0,Y 387.352,Z 572.854,A -85,B 0,C 180,E1 -11951.9,E2 -11951.9} C_VEL
LIN {X 0,Y 386.252,Z 582.537,A -85,B 0,C 180,E1 -11953.076,E2 -11953.076} C_VEL
LIN {X 0,Y 384.984,Z 593.266,A -85,B 0,C 180,E1 -11954.653,E2 -11954.653} C_VEL
LIN {X 0,Y 384.017,Z 602.125,A -85,B 0,C 180,E1 -11956.238,E2 -11956.238} C_VEL
LIN {X 0,Y 383.273,Z 609.498,A -85,B 0,C 180,E1 -11957.828,E2 -11957.828} C_VEL
LIN {X 0,Y 382.553,Z 615.641,A -85,B 0,C 180,E1 -11959.416,E2 -11959.416} C_VEL
LIN {X 0,Y 382.157,Z 620.731,A -85,B 0,C 180,E1 -11961.008,E2 -11961.008} C_VEL
LIN {X 0,Y 381.78,Z 625.989,A -85,B 0,C 180,E1 -11963.129,E2 -11963.129} C_VEL
LIN {X 0,Y 381.648,Z 628.934,A -85,B 0,C 180,E1 -11964.719,E2 -11964.719} C_VEL
LIN {X 0,Y 381.509,Z 631.625,A -85,B 0,C 180,E1 -11966.834,E2 -11966.834} C_VEL
LIN {X 0,Y 381.551,Z 632.955,A -85,B 0,C 180,E1 -11968.946,E2 -11968.946} C_VEL
LIN {X 0,Y 381.551,Z 632.951,A -85,B 0,C 180,E1 -11971.057,E2 -11971.057} C_VEL
LIN {X 0,Y 381.51,Z 631.61,A -85,B 0,C 180,E1 -11973.17,E2 -11973.17} C_VEL
LIN {X 0,Y 381.648,Z 628.911,A -85,B 0,C 180,E1 -11975.284,E2 -11975.284} C_VEL
LIN {X 0,Y 381.793,Z 625.964,A -85,B 0,C 180,E1 -11976.873,E2 -11976.873} C_VEL
LIN {X 0,Y 382.16,Z 620.7,A -85,B 0,C 180,E1 -11978.995,E2 -11978.995} C_VEL
LIN {X 0,Y 382.557,Z 615.601,A -85,B 0,C 180,E1 -11980.587,E2 -11980.587} C_VEL
LIN {X 0,Y 383.406,Z 608.329,A -85,B 0,C 180,E1 -11982.439,E2 -11982.439} C_VEL
LIN {X 0,Y 384.233,Z 599.81,A -85,B 0,C 180,E1 -11984.205,E2 -11984.205} C_VEL
LIN {X 0,Y 385.387,Z 589.867,A -85,B 0,C 180,E1 -11985.877,E2 -11985.877} C_VEL
LIN {X 0,Y 386.612,Z 579.404,A -85,B 0,C 180,E1 -11987.319,E2 -11987.319} C_VEL
LIN {X 0,Y 387.919,Z 567.852,A -85,B 0,C 180,E1 -11988.623,E2 -11988.623} C_VEL
LIN {X 0,Y 389.252,Z 555.034,A -85,B 0,C 180,E1 -11989.789,E2 -11989.789} C_VEL
LIN {X 0,Y 390.33,Z 542.261,A -85,B 0,C 180,E1 -11990.712,E2 -11990.712} C_VEL
LIN {X 0,Y 391.271,Z 528.582,A -85,B 0,C 180,E1 -11991.469,E2 -11991.469} C_VEL
LIN {X 0,Y 392.11,Z 514.813,A -85,B 0,C 180,E1 -11992.008,E2 -11992.008} C_VEL
LIN {X 0,Y 392.581,Z 500.715,A -85,B 0,C 180,E1 -11992.361,E2 -11992.361} C_VEL
LIN {X 0,Y 394.342,Z 404.73,A -85,B 0,C 180,E1 -11994.118,E2 -11994.118} C_VEL
LIN {X 0,Y 393.952,Z 400.502,A -85,B 0,C 180,E1 -11994.226,E2 -11994.226} C_VEL
LIN {X 0,Y 388.165,Z 371.649,A -85,B 0,C 180,E1 -11995.185,E2 -11995.185} C_VEL
LIN {X 0,Y 387.93,Z 370.259,A -85,B 0,C 180,E1 -11995.253,E2 -11995.253} C_VEL
LIN {X 0,Y 387.198,Z 365.148,A -85,B 0,C 180,E1 -11996.405,E2 -11996.405} C_VEL
LIN {X 0,Y 384.566,Z 352.745,A -85,B 0,C 180,E1 -11999.338,E2 -11999.338} C_VEL
LIN {X 0,Y 383.007,Z 346.402,A -85,B 0,C 180,E1 -12000.918,E2 -12000.918} C_VEL
LIN {X 0,Y 383.023,Z 346.397,A -85,B 0,C 180,E1 -12004.669,E2 -12004.669} C_VEL
LIN {X 0,Y 383.003,Z 346.399,A -85,B 0,C 180,E1 -12007.904,E2 -12007.904} C_VEL
LIN {X 0,Y 382.989,Z 346.404,A -85,B 0,C 180,E1 -12011.348,E2 -12011.348} C_VEL
LIN {X 0,Y 383.001,Z 346.399,A -85,B 0,C 180,E1 -12014.304,E2 -12014.304} C_VEL
LIN {X 0,Y 383.016,Z 346.401,A -85,B 0,C 180,E1 -12017.241,E2 -12017.241} C_VEL
LIN {X 0,Y 383.021,Z 346.398,A -85,B 0,C 180,E1 -12020.414,E2 -12020.414} C_VEL
LIN {X 0,Y 383.03,Z 346.398,A -85,B 0,C 180,E1 -12024.045,E2 -12024.045} C_VEL
LIN {X 0,Y 382.992,Z 346.406,A -85,B 0,C 180,E1 -12027.579,E2 -12027.579} C_VEL
LIN {X 0,Y 383.004,Z 346.446,A -85,B 0,C 180,E1 -12029.389,E2 -12029.389} C_VEL
LIN {X 0,Y 385.986,Z 355.283,A -85,B 0,C 180,E1 -12031.744,E2 -12031.744} C_VEL
LIN {X 0,Y 388.587,Z 364.49,A -85,B 0,C 180,E1 -12034,E2 -12034} C_VEL
LIN {X 0,Y 389.857,Z 371.111,A -85,B 0,C 180,E1 -12035.504,E2 -12035.504} C_VEL
LIN {X 0,Y 389.813,Z 376.763,A -85,B 0,C 180,E1 -12036.632,E2 -12036.632} C_VEL
LIN {X 0,Y 389.539,Z 382.504,A -85,B 0,C 180,E1 -12037.706,E2 -12037.706} C_VEL
LIN {X 0,Y 392.943,Z 396.152,A -85,B 0,C 180,E1 -12038.496,E2 -12038.496} C_VEL
LIN {X 0,Y 394.128,Z 403.129,A -85,B 0,C 180,E1 -12038.832,E2 -12038.832} C_VEL
LIN {X 0,Y 390.835,Z 480.687,A -85,B 0,C 180,E1 -12040.91,E2 -12040.91} C_VEL
LIN {X 0,Y 390.236,Z 495.467,A -85,B 0,C 180,E1 -12041.357,E2 -12041.357} C_VEL
LIN {X 0,Y 389.527,Z 509.354,A -85,B 0,C 180,E1 -12042.003,E2 -12042.003} C_VEL
LIN {X 0,Y 388.743,Z 521.417,A -85,B 0,C 180,E1 -12042.78,E2 -12042.78} C_VEL
LIN {X 0,Y 387.772,Z 533.083,A -85,B 0,C 180,E1 -12043.739,E2 -12043.739} C_VEL
LIN {X 0,Y 386.775,Z 543.953,A -85,B 0,C 180,E1 -12044.87,E2 -12044.87} C_VEL
LIN {X 0,Y 385.576,Z 554.963,A -85,B 0,C 180,E1 -12046.293,E2 -12046.293} C_VEL
LIN {X 0,Y 384.622,Z 564.527,A -85,B 0,C 180,E1 -12047.87,E2 -12047.87} C_VEL
LIN {X 0,Y 383.848,Z 572.224,A -85,B 0,C 180,E1 -12049.45,E2 -12049.45} C_VEL
LIN {X 0,Y 383.093,Z 578.352,A -85,B 0,C 180,E1 -12051.029,E2 -12051.029} C_VEL
LIN {X 0,Y 382.642,Z 583.34,A -85,B 0,C 180,E1 -12052.674,E2 -12052.674} C_VEL
LIN {X 0,Y 382.176,Z 586.849,A -85,B 0,C 180,E1 -12054.195,E2 -12054.195} C_VEL
LIN {X 0,Y 382.069,Z 589.429,A -85,B 0,C 180,E1 -12055.781,E2 -12055.781} C_VEL
LIN {X 0,Y 381.977,Z 590.618,A -85,B 0,C 180,E1 -12056.836,E2 -12056.836} C_VEL
LIN {X 0,Y 381.817,Z 591.349,A -85,B 0,C 180,E1 -12057.89,E2 -12057.89} C_VEL
LIN {X 0,Y 381.72,Z 591.639,A -85,B 0,C 180,E1 -12058.945,E2 -12058.945} C_VEL
LIN {X 0,Y 381.68,Z 591.519,A -85,B 0,C 180,E1 -12060,E2 -12060} C_VEL
LIN {X 0,Y 381.7,Z 590.95,A -85,B 0,C 180,E1 -12061.055,E2 -12061.055} C_VEL
LIN {X 0,Y 381.754,Z 589.929,A -85,B 0,C 180,E1 -12062.11,E2 -12062.11} C_VEL
LIN {X 0,Y 381.758,Z 588.496,A -85,B 0,C 180,E1 -12063.166,E2 -12063.166} C_VEL
LIN {X 0,Y 381.866,Z 585.467,A -85,B 0,C 180,E1 -12064.751,E2 -12064.751} C_VEL
LIN {X 0,Y 382.042,Z 581.333,A -85,B 0,C 180,E1 -12066.337,E2 -12066.337} C_VEL
LIN {X 0,Y 382.333,Z 574.912,A -85,B 0,C 180,E1 -12068.19,E2 -12068.19} C_VEL
LIN {X 0,Y 382.762,Z 567.9,A -85,B 0,C 180,E1 -12069.779,E2 -12069.779} C_VEL
LIN {X 0,Y 383.21,Z 560.728,A -85,B 0,C 180,E1 -12071.103,E2 -12071.103} C_VEL
LIN {X 0,Y 383.787,Z 552.032,A -85,B 0,C 180,E1 -12072.426,E2 -12072.426} C_VEL
LIN {X 0,Y 384.496,Z 541.393,A -85,B 0,C 180,E1 -12073.746,E2 -12073.746} C_VEL
LIN {X 0,Y 385.071,Z 530.886,A -85,B 0,C 180,E1 -12074.804,E2 -12074.804} C_VEL
LIN {X 0,Y 385.648,Z 519.343,A -85,B 0,C 180,E1 -12075.729,E2 -12075.729} C_VEL
LIN {X 0,Y 386.304,Z 506.645,A -85,B 0,C 180,E1 -12076.515,E2 -12076.515} C_VEL
LIN {X 0,Y 386.734,Z 493.283,A -85,B 0,C 180,E1 -12077.108,E2 -12077.108} C_VEL
LIN {X 0,Y 387.088,Z 479.598,A -85,B 0,C 180,E1 -12077.5,E2 -12077.5} C_VEL
LIN {X 0,Y 388.783,Z 399.27,A -85,B 0,C 180,E1 -12079.37,E2 -12079.37} C_VEL
LIN {X 0,Y 385.464,Z 378.414,A -85,B 0,C 180,E1 -12080.019,E2 -12080.019} C_VEL
LIN {X 0,Y 386.081,Z 362.448,A -85,B 0,C 180,E1 -12083.04,E2 -12083.04} C_VEL
LIN {X 0,Y 383.88,Z 350.327,A -85,B 0,C 180,E1 -12085.483,E2 -12085.483} C_VEL
LIN {X 0,Y 383.087,Z 346.394,A -85,B 0,C 180,E1 -12086.306,E2 -12086.306} C_VEL
LIN {X 0,Y 382.998,Z 346.402,A -85,B 0,C 180,E1 -12089.7,E2 -12089.7} C_VEL
LIN {X 0,Y 383.01,Z 346.399,A -85,B 0,C 180,E1 -12093.4,E2 -12093.4} C_VEL
LIN {X 0,Y 383.037,Z 346.397,A -85,B 0,C 180,E1 -12096.164,E2 -12096.164} C_VEL
LIN {X 0,Y 382.981,Z 346.407,A -85,B 0,C 180,E1 -12099.962,E2 -12099.962} C_VEL
LIN {X 0,Y 383.012,Z 346.399,A -85,B 0,C 180,E1 -12102.778,E2 -12102.778} C_VEL
LIN {X 0,Y 383.001,Z 346.406,A -85,B 0,C 180,E1 -12105.788,E2 -12105.788} C_VEL
LIN {X 0,Y 382.967,Z 346.404,A -85,B 0,C 180,E1 -12108.8,E2 -12108.8} C_VEL
LIN {X 0,Y 382.997,Z 346.403,A -85,B 0,C 180,E1 -12112.097,E2 -12112.097} C_VEL
LIN {X 0,Y 383.016,Z 346.397,A -85,B 0,C 180,E1 -12115.33,E2 -12115.33} C_VEL
LIN {X 0,Y 382.983,Z 346.404,A -85,B 0,C 180,E1 -12119.08,E2 -12119.08} C_VEL
LIN {X 0,Y 383.049,Z 346.499,A -85,B 0,C 180,E1 -12120.417,E2 -12120.417} C_VEL
LIN {X 0,Y 385.988,Z 359.597,A -85,B 0,C 180,E1 -12123.696,E2 -12123.696} C_VEL
LIN {X 0,Y 386.901,Z 364.223,A -85,B 0,C 180,E1 -12124.756,E2 -12124.756} C_VEL
LIN {X 0,Y 389.988,Z 372.141,A -85,B 0,C 180,E1 -12125.128,E2 -12125.128} C_VEL
LIN {X 0,Y 394.467,Z 394.289,A -85,B 0,C 180,E1 -12125.864,E2 -12125.864} C_VEL
LIN {X 0,Y 392.532,Z 499.456,A -85,B 0,C 180,E1 -12127.809,E2 -12127.809} C_VEL
LIN {X 0,Y 391.923,Z 514.017,A -85,B 0,C 180,E1 -12128.258,E2 -12128.258} C_VEL
LIN {X 0,Y 391.098,Z 527.277,A -85,B 0,C 180,E1 -12128.866,E2 -12128.866} C_VEL
LIN {X 0,Y 390.118,Z 540.4,A -85,B 0,C 180,E1 -12129.68,E2 -12129.68} C_VEL
LIN {X 0,Y 389.04,Z 552.239,A -85,B 0,C 180,E1 -12130.612,E2 -12130.612} C_VEL
LIN {X 0,Y 387.802,Z 564.205,A -85,B 0,C 180,E1 -12131.782,E2 -12131.782} C_VEL
LIN {X 0,Y 386.559,Z 575.119,A -85,B 0,C 180,E1 -12133.087,E2 -12133.087} C_VEL
LIN {X 0,Y 385.235,Z 585.884,A -85,B 0,C 180,E1 -12134.66,E2 -12134.66} C_VEL
LIN {X 0,Y 384.322,Z 594.767,A -85,B 0,C 180,E1 -12136.246,E2 -12136.246} C_VEL
LIN {X 0,Y 383.299,Z 603.273,A -85,B 0,C 180,E1 -12138.094,E2 -12138.094} C_VEL
LIN {X 0,Y 382.704,Z 609.251,A -85,B 0,C 180,E1 -12139.692,E2 -12139.692} C_VEL
LIN {X 0,Y 381.788,Z 611.868,A -85,B 0,C 180,E1 -12140.475,E2 -12140.475} C_VEL
LIN {X 0,Y 377.228,Z 617.089,A -85,B 0,C 180,E1 -12142.293,E2 -12142.293} C_VEL
LIN {X 0,Y 375.117,Z 619.539,A -85,B 0,C 180,E1 -12143.397,E2 -12143.397} C_VEL
LIN {X 0,Y 374.725,Z 620.6,A -85,B 0,C 180,E1 -12143.975,E2 -12143.975} C_VEL
LIN {X 0,Y 374.579,Z 623.228,A -85,B 0,C 180,E1 -12145.694,E2 -12145.694} C_VEL
LIN {X 0,Y 374.457,Z 625.257,A -85,B 0,C 180,E1 -12147.847,E2 -12147.847} C_VEL
LIN {X 0,Y 374.473,Z 625.954,A -85,B 0,C 180,E1 -12149.998,E2 -12149.998} C_VEL
LIN {X 0,Y 374.456,Z 625.33,A -85,B 0,C 180,E1 -12152.15,E2 -12152.15} C_VEL
LIN {X 0,Y 374.575,Z 623.37,A -85,B 0,C 180,E1 -12154.302,E2 -12154.302} C_VEL
LIN {X 0,Y 374.726,Z 620.024,A -85,B 0,C 180,E1 -12156.459,E2 -12156.459} C_VEL
LIN {X 0,Y 375.115,Z 615.192,A -85,B 0,C 180,E1 -12158.618,E2 -12158.618} C_VEL
LIN {X 0,Y 375.763,Z 608.731,A -85,B 0,C 180,E1 -12160.778,E2 -12160.778} C_VEL
LIN {X 0,Y 376.613,Z 601.536,A -85,B 0,C 180,E1 -12162.664,E2 -12162.664} C_VEL
LIN {X 0,Y 377.438,Z 593.902,A -85,B 0,C 180,E1 -12164.301,E2 -12164.301} C_VEL
LIN {X 0,Y 378.525,Z 584.94,A -85,B 0,C 180,E1 -12165.892,E2 -12165.892} C_VEL
LIN {X 0,Y 379.929,Z 573.968,A -85,B 0,C 180,E1 -12167.491,E2 -12167.491} C_VEL
LIN {X 0,Y 381.246,Z 562.783,A -85,B 0,C 180,E1 -12168.818,E2 -12168.818} C_VEL
LIN {X 0,Y 382.579,Z 550.408,A -85,B 0,C 180,E1 -12170.005,E2 -12170.005} C_VEL
LIN {X 0,Y 383.713,Z 537.218,A -85,B 0,C 180,E1 -12171.013,E2 -12171.013} C_VEL
LIN {X 0,Y 384.787,Z 522.829,A -85,B 0,C 180,E1 -12171.846,E2 -12171.846} C_VEL
LIN {X 0,Y 385.611,Z 508.608,A -85,B 0,C 180,E1 -12172.431,E2 -12172.431} C_VEL
LIN {X 0,Y 386.174,Z 494.984,A -85,B 0,C 180,E1 -12172.785,E2 -12172.785} C_VEL
LIN {X 0,Y 387.993,Z 395.036,A -85,B 0,C 180,E1 -12174.654,E2 -12174.654} C_VEL
LIN {X 0,Y 383.431,Z 373.425,A -85,B 0,C 180,E1 -12175.406,E2 -12175.406} C_VEL
LIN {X 0,Y 379.636,Z 363.952,A -85,B 0,C 180,E1 -12175.892,E2 -12175.892} C_VEL
LIN {X 0,Y 376.994,Z 351.641,A -85,B 0,C 180,E1 -12178.99,E2 -12178.99} C_VEL
LIN {X 0,Y 375.973,Z 347.282,A -85,B 0,C 180,E1 -12180.155,E2 -12180.155} C_VEL
LIN {X 0,Y 375.954,Z 347.283,A -85,B 0,C 180,E1 -12184.11,E2 -12184.11} C_VEL
LIN {X 0,Y 375.945,Z 347.284,A -85,B 0,C 180,E1 -12186.74,E2 -12186.74} C_VEL
LIN {X 0,Y 375.93,Z 347.281,A -85,B 0,C 180,E1 -12189.96,E2 -12189.96} C_VEL
LIN {X 0,Y 375.916,Z 347.282,A -85,B 0,C 180,E1 -12193.765,E2 -12193.765} C_VEL
LIN {X 0,Y 375.924,Z 347.283,A -85,B 0,C 180,E1 -12196.809,E2 -12196.809} C_VEL
LIN {X 0,Y 375.924,Z 347.284,A -85,B 0,C 180,E1 -12200.532,E2 -12200.532} C_VEL
LIN {X 0,Y 375.951,Z 347.278,A -85,B 0,C 180,E1 -12203.495,E2 -12203.495} C_VEL
LIN {X 0,Y 375.947,Z 347.275,A -85,B 0,C 180,E1 -12205.887,E2 -12205.887} C_VEL
LIN {X 0,Y 375.949,Z 347.277,A -85,B 0,C 180,E1 -12209.686,E2 -12209.686} C_VEL
LIN {X 0,Y 375.905,Z 347.281,A -85,B 0,C 180,E1 -12212.134,E2 -12212.134} C_VEL
LIN {X 0,Y 375.946,Z 347.276,A -85,B 0,C 180,E1 -12215.715,E2 -12215.715} C_VEL
LIN {X 0,Y 375.966,Z 347.266,A -85,B 0,C 180,E1 -12219.196,E2 -12219.196} C_VEL
LIN {X 0,Y 376.018,Z 347.261,A -85,B 0,C 180,E1 -12222.599,E2 -12222.599} C_VEL
LIN {X 0,Y 376.076,Z 347.263,A -85,B 0,C 180,E1 -12226.342,E2 -12226.342} C_VEL
LIN {X 0,Y 376.098,Z 347.261,A -85,B 0,C 180,E1 -12230.318,E2 -12230.318} C_VEL
LIN {X 0,Y 376.174,Z 347.249,A -85,B 0,C 180,E1 -12233.564,E2 -12233.564} C_VEL
LIN {X 0,Y 376.326,Z 347.231,A -85,B 0,C 180,E1 -12237.859,E2 -12237.859} C_VEL
LIN {X 0,Y 376.323,Z 347.233,A -85,B 0,C 180,E1 -12242.14,E2 -12242.14} C_VEL
LIN {X 0,Y 376.184,Z 347.253,A -85,B 0,C 180,E1 -12246.436,E2 -12246.436} C_VEL
LIN {X 0,Y 376.092,Z 347.258,A -85,B 0,C 180,E1 -12249.682,E2 -12249.682} C_VEL
LIN {X 0,Y 376.075,Z 347.259,A -85,B 0,C 180,E1 -12253.658,E2 -12253.658} C_VEL
LIN {X 0,Y 376.018,Z 347.266,A -85,B 0,C 180,E1 -12257.4,E2 -12257.4} C_VEL
LIN {X 0,Y 375.965,Z 347.267,A -85,B 0,C 180,E1 -12260.833,E2 -12260.833} C_VEL
LIN {X 0,Y 375.921,Z 347.277,A -85,B 0,C 180,E1 -12264.286,E2 -12264.286} C_VEL
LIN {X 0,Y 375.899,Z 347.284,A -85,B 0,C 180,E1 -12266.661,E2 -12266.661} C_VEL
LIN {X 0,Y 375.9,Z 347.271,A -85,B 0,C 180,E1 -12269.085,E2 -12269.085} C_VEL
LIN {X 0,Y 375.925,Z 347.281,A -85,B 0,C 180,E1 -12271.565,E2 -12271.565} C_VEL
LIN {X 0,Y 375.962,Z 347.279,A -85,B 0,C 180,E1 -12274.667,E2 -12274.667} C_VEL
LIN {X 0,Y 375.922,Z 347.284,A -85,B 0,C 180,E1 -12278.264,E2 -12278.264} C_VEL
LIN {X 0,Y 375.901,Z 347.284,A -85,B 0,C 180,E1 -12281.598,E2 -12281.598} C_VEL
LIN {X 0,Y 375.909,Z 347.286,A -85,B 0,C 180,E1 -12284.732,E2 -12284.732} C_VEL
LIN {X 0,Y 375.897,Z 347.288,A -85,B 0,C 180,E1 -12287.698,E2 -12287.698} C_VEL
LIN {X 0,Y 375.923,Z 347.287,A -85,B 0,C 180,E1 -12290.535,E2 -12290.535} C_VEL
LIN {X 0,Y 375.948,Z 347.282,A -85,B 0,C 180,E1 -12293.499,E2 -12293.499} C_VEL
LIN {X 0,Y 375.95,Z 347.283,A -85,B 0,C 180,E1 -12295.89,E2 -12295.89} C_VEL
LIN {X 0,Y 375.957,Z 347.334,A -85,B 0,C 180,E1 -12298.668,E2 -12298.668} C_VEL
LIN {X 0,Y 378.872,Z 359.796,A -85,B 0,C 180,E1 -12301.772,E2 -12301.772} C_VEL
LIN {X 0,Y 381.083,Z 370.543,A -85,B 0,C 180,E1 -12304.279,E2 -12304.279} C_VEL
LIN {X 0,Y 385.025,Z 388.501,A -85,B 0,C 180,E1 -12304.923,E2 -12304.923} C_VEL
LIN {X 0,Y 387.854,Z 403.781,A -85,B 0,C 180,E1 -12305.423,E2 -12305.423} C_VEL
LIN {X 0,Y 385.898,Z 507.312,A -85,B 0,C 180,E1 -12307.375,E2 -12307.375} C_VEL
LIN {X 0,Y 385.182,Z 521.392,A -85,B 0,C 180,E1 -12307.825,E2 -12307.825} C_VEL
LIN {X 0,Y 384.264,Z 535.075,A -85,B 0,C 180,E1 -12308.475,E2 -12308.475} C_VEL
LIN {X 0,Y 383.19,Z 547.887,A -85,B 0,C 180,E1 -12309.29,E2 -12309.29} C_VEL
LIN {X 0,Y 381.939,Z 561.161,A -85,B 0,C 180,E1 -12310.38,E2 -12310.38} C_VEL
LIN {X 0,Y 380.594,Z 572.79,A -85,B 0,C 180,E1 -12311.567,E2 -12311.567} C_VEL
LIN {X 0,Y 379.418,Z 582.472,A -85,B 0,C 180,E1 -12312.762,E2 -12312.762} C_VEL
LIN {X 0,Y 378.088,Z 593.201,A -85,B 0,C 180,E1 -12314.366,E2 -12314.366} C_VEL
LIN {X 0,Y 377.088,Z 602.059,A -85,B 0,C 180,E1 -12315.98,E2 -12315.98} C_VEL
LIN {X 0,Y 376.183,Z 610.55,A -85,B 0,C 180,E1 -12317.869,E2 -12317.869} C_VEL
LIN {X 0,Y 375.374,Z 617.387,A -85,B 0,C 180,E1 -12319.756,E2 -12319.756} C_VEL
LIN {X 0,Y 374.977,Z 622.101,A -85,B 0,C 180,E1 -12321.378,E2 -12321.378} C_VEL
LIN {X 0,Y 374.629,Z 626.99,A -85,B 0,C 180,E1 -12323.539,E2 -12323.539} C_VEL
LIN {X 0,Y 374.515,Z 630.386,A -85,B 0,C 180,E1 -12325.697,E2 -12325.697} C_VEL
LIN {X 0,Y 374.41,Z 632.391,A -85,B 0,C 180,E1 -12327.85,E2 -12327.85} C_VEL
LIN {X 0,Y 374.472,Z 633.052,A -85,B 0,C 180,E1 -12330.002,E2 -12330.002} C_VEL
LIN {X 0,Y 374.411,Z 632.38,A -85,B 0,C 180,E1 -12332.153,E2 -12332.153} C_VEL
LIN {X 0,Y 374.514,Z 630.366,A -85,B 0,C 180,E1 -12334.306,E2 -12334.306} C_VEL
LIN {X 0,Y 374.678,Z 626.963,A -85,B 0,C 180,E1 -12336.464,E2 -12336.464} C_VEL
LIN {X 0,Y 374.98,Z 622.07,A -85,B 0,C 180,E1 -12338.625,E2 -12338.625} C_VEL
LIN {X 0,Y 375.532,Z 615.532,A -85,B 0,C 180,E1 -12340.788,E2 -12340.788} C_VEL
LIN {X 0,Y 376.444,Z 608.26,A -85,B 0,C 180,E1 -12342.673,E2 -12342.673} C_VEL
LIN {X 0,Y 377.364,Z 599.259,A -85,B 0,C 180,E1 -12344.562,E2 -12344.562} C_VEL
LIN {X 0,Y 378.518,Z 589.797,A -85,B 0,C 180,E1 -12346.173,E2 -12346.173} C_VEL
LIN {X 0,Y 379.805,Z 579.333,A -85,B 0,C 180,E1 -12347.64,E2 -12347.64} C_VEL
LIN {X 0,Y 381.154,Z 567.781,A -85,B 0,C 180,E1 -12348.966,E2 -12348.966} C_VEL
LIN {X 0,Y 382.578,Z 554.963,A -85,B 0,C 180,E1 -12350.149,E2 -12350.149} C_VEL
LIN {X 0,Y 383.74,Z 541.586,A -85,B 0,C 180,E1 -12351.127,E2 -12351.127} C_VEL
LIN {X 0,Y 384.68,Z 528.507,A -85,B 0,C 180,E1 -12351.856,E2 -12351.856} C_VEL
LIN {X 0,Y 385.541,Z 514.735,A -85,B 0,C 180,E1 -12352.403,E2 -12352.403} C_VEL
LIN {X 0,Y 386.036,Z 500.628,A -85,B 0,C 180,E1 -12352.761,E2 -12352.761} C_VEL
LIN {X 0,Y 387.886,Z 404.643,A -85,B 0,C 180,E1 -12354.546,E2 -12354.546} C_VEL
LIN {X 0,Y 383.561,Z 381.356,A -85,B 0,C 180,E1 -12355.311,E2 -12355.311} C_VEL
LIN {X 0,Y 381.057,Z 370.485,A -85,B 0,C 180,E1 -12355.711,E2 -12355.711} C_VEL
LIN {X 0,Y 378.58,Z 358.371,A -85,B 0,C 180,E1 -12358.558,E2 -12358.558} C_VEL
LIN {X 0,Y 375.96,Z 347.278,A -85,B 0,C 180,E1 -12361.332,E2 -12361.332} C_VEL
LIN {X 0,Y 375.985,Z 347.273,A -85,B 0,C 180,E1 -12364.668,E2 -12364.668} C_VEL
LIN {X 0,Y 375.978,Z 347.273,A -85,B 0,C 180,E1 -12368.271,E2 -12368.271} C_VEL
LIN {X 0,Y 375.94,Z 347.281,A -85,B 0,C 180,E1 -12371.602,E2 -12371.602} C_VEL
LIN {X 0,Y 375.932,Z 347.284,A -85,B 0,C 180,E1 -12375.269,E2 -12375.269} C_VEL
LIN {X 0,Y 375.94,Z 347.279,A -85,B 0,C 180,E1 -12378.4,E2 -12378.4} C_VEL
LIN {X 0,Y 375.979,Z 347.274,A -85,B 0,C 180,E1 -12381.73,E2 -12381.73} C_VEL
LIN {X 0,Y 375.985,Z 347.275,A -85,B 0,C 180,E1 -12385.333,E2 -12385.333} C_VEL
LIN {X 0,Y 375.969,Z 347.377,A -85,B 0,C 180,E1 -12388.367,E2 -12388.367} C_VEL
LIN {X 0,Y 379.457,Z 357.357,A -85,B 0,C 180,E1 -12391.213,E2 -12391.213} C_VEL
LIN {X 0,Y 382.076,Z 366.568,A -85,B 0,C 180,E1 -12393.549,E2 -12393.549} C_VEL
LIN {X 0,Y 383.554,Z 374.321,A -85,B 0,C 180,E1 -12395.364,E2 -12395.364} C_VEL
LIN {X 0,Y 383.222,Z 382.924,A -85,B 0,C 180,E1 -12397.058,E2 -12397.058} C_VEL
LIN {X 0,Y 386.787,Z 396.961,A -85,B 0,C 180,E1 -12397.925,E2 -12397.925} C_VEL
LIN {X 0,Y 388.09,Z 403.494,A -85,B 0,C 180,E1 -12398.277,E2 -12398.277} C_VEL
LIN {X 0,Y 384.609,Z 479.099,A -85,B 0,C 180,E1 -12400.381,E2 -12400.381} C_VEL
LIN {X 0,Y 383.914,Z 495.138,A -85,B 0,C 180,E1 -12400.865,E2 -12400.865} C_VEL
LIN {X 0,Y 383.178,Z 508.511,A -85,B 0,C 180,E1 -12401.486,E2 -12401.486} C_VEL
LIN {X 0,Y 382.378,Z 519.972,A -85,B 0,C 180,E1 -12402.208,E2 -12402.208} C_VEL
LIN {X 0,Y 381.264,Z 533.208,A -85,B 0,C 180,E1 -12403.302,E2 -12403.302} C_VEL
LIN {X 0,Y 380.216,Z 543.495,A -85,B 0,C 180,E1 -12404.373,E2 -12404.373} C_VEL
LIN {X 0,Y 379.051,Z 554.31,A -85,B 0,C 180,E1 -12405.779,E2 -12405.779} C_VEL
LIN {X 0,Y 378.135,Z 562.638,A -85,B 0,C 180,E1 -12407.113,E2 -12407.113} C_VEL
LIN {X 0,Y 377.14,Z 570.744,A -85,B 0,C 180,E1 -12408.716,E2 -12408.716} C_VEL
LIN {X 0,Y 376.364,Z 577.265,A -85,B 0,C 180,E1 -12410.325,E2 -12410.325} C_VEL
LIN {X 0,Y 375.803,Z 582.436,A -85,B 0,C 180,E1 -12411.937,E2 -12411.937} C_VEL
LIN {X 0,Y 375.344,Z 586.388,A -85,B 0,C 180,E1 -12413.55,E2 -12413.55} C_VEL
LIN {X 0,Y 374.998,Z 588.397,A -85,B 0,C 180,E1 -12414.623,E2 -12414.623} C_VEL
LIN {X 0,Y 375.006,Z 589.953,A -85,B 0,C 180,E1 -12415.701,E2 -12415.701} C_VEL
LIN {X 0,Y 374.924,Z 591.089,A -85,B 0,C 180,E1 -12416.776,E2 -12416.776} C_VEL
LIN {X 0,Y 374.758,Z 591.756,A -85,B 0,C 180,E1 -12417.851,E2 -12417.851} C_VEL
LIN {X 0,Y 374.654,Z 592.007,A -85,B 0,C 180,E1 -12418.925,E2 -12418.925} C_VEL
LIN {X 0,Y 374.612,Z 591.841,A -85,B 0,C 180,E1 -12420,E2 -12420} C_VEL
LIN {X 0,Y 374.634,Z 591.199,A -85,B 0,C 180,E1 -12421.075,E2 -12421.075} C_VEL
LIN {X 0,Y 374.657,Z 590.134,A -85,B 0,C 180,E1 -12422.15,E2 -12422.15} C_VEL
LIN {X 0,Y 374.662,Z 588.653,A -85,B 0,C 180,E1 -12423.226,E2 -12423.226} C_VEL
LIN {X 0,Y 374.802,Z 585.528,A -85,B 0,C 180,E1 -12424.841,E2 -12424.841} C_VEL
LIN {X 0,Y 375.038,Z 580.079,A -85,B 0,C 180,E1 -12426.839,E2 -12426.839} C_VEL
LIN {X 0,Y 375.34,Z 573.657,A -85,B 0,C 180,E1 -12428.615,E2 -12428.615} C_VEL
LIN {X 0,Y 375.846,Z 566.19,A -85,B 0,C 180,E1 -12430.233,E2 -12430.233} C_VEL
LIN {X 0,Y 376.411,Z 556.91,A -85,B 0,C 180,E1 -12431.852,E2 -12431.852} C_VEL
LIN {X 0,Y 377.206,Z 546.231,A -85,B 0,C 180,E1 -12433.331,E2 -12433.331} C_VEL
LIN {X 0,Y 377.815,Z 535.481,A -85,B 0,C 180,E1 -12434.534,E2 -12434.534} C_VEL
LIN {X 0,Y 378.485,Z 523.22,A -85,B 0,C 180,E1 -12435.62,E2 -12435.62} C_VEL
LIN {X 0,Y 379.091,Z 510.425,A -85,B 0,C 180,E1 -12436.492,E2 -12436.492} C_VEL
LIN {X 0,Y 379.676,Z 497.074,A -85,B 0,C 180,E1 -12437.158,E2 -12437.158} C_VEL
LIN {X 0,Y 380.062,Z 484.133,A -85,B 0,C 180,E1 -12437.591,E2 -12437.591} C_VEL
LIN {X 0,Y 381.858,Z 399.834,A -85,B 0,C 180,E1 -12439.617,E2 -12439.617} C_VEL
LIN {X 0,Y 378.504,Z 378.581,A -85,B 0,C 180,E1 -12440.308,E2 -12440.308} C_VEL
LIN {X 0,Y 379.102,Z 363.429,A -85,B 0,C 180,E1 -12443.2,E2 -12443.2} C_VEL
LIN {X 0,Y 376.642,Z 350.204,A -85,B 0,C 180,E1 -12445.896,E2 -12445.896} C_VEL
LIN {X 0,Y 376.06,Z 347.269,A -85,B 0,C 180,E1 -12446.519,E2 -12446.519} C_VEL
LIN {X 0,Y 375.971,Z 347.277,A -85,B 0,C 180,E1 -12450.312,E2 -12450.312} C_VEL
LIN {X 0,Y 375.966,Z 347.279,A -85,B 0,C 180,E1 -12454.111,E2 -12454.111} C_VEL
LIN {X 0,Y 375.958,Z 347.277,A -85,B 0,C 180,E1 -12456.741,E2 -12456.741} C_VEL
LIN {X 0,Y 375.944,Z 347.283,A -85,B 0,C 180,E1 -12459.961,E2 -12459.961} C_VEL
LIN {X 0,Y 375.935,Z 347.285,A -85,B 0,C 180,E1 -12463.765,E2 -12463.765} C_VEL
LIN {X 0,Y 375.939,Z 347.28,A -85,B 0,C 180,E1 -12466.81,E2 -12466.81} C_VEL
LIN {X 0,Y 375.939,Z 347.28,A -85,B 0,C 180,E1 -12470.533,E2 -12470.533} C_VEL
LIN {X 0,Y 375.963,Z 347.28,A -85,B 0,C 180,E1 -12473.496,E2 -12473.496} C_VEL
LIN {X 0,Y 375.962,Z 347.279,A -85,B 0,C 180,E1 -12475.887,E2 -12475.887} C_VEL
LIN {X 0,Y 375.981,Z 347.276,A -85,B 0,C 180,E1 -12479.842,E2 -12479.842} C_VEL
LIN {X 0,Y 375.99,Z 347.363,A -85,B 0,C 180,E1 -12479.998,E2 -12479.998} C_VEL
LIN {X 0,Y 378.615,Z 359.055,A -85,B 0,C 180,E1 -12482.999,E2 -12482.999} C_VEL
LIN {X 0,Y 379.723,Z 364.289,A -85,B 0,C 180,E1 -12484.243,E2 -12484.243} C_VEL
LIN {X 0,Y 384.016,Z 375.487,A -85,B 0,C 180,E1 -12484.78,E2 -12484.78} C_VEL
LIN {X 0,Y 388.015,Z 395.978,A -85,B 0,C 180,E1 -12485.469,E2 -12485.469} C_VEL
LIN {X 0,Y 385.946,Z 500.957,A -85,B 0,C 180,E1 -12487.445,E2 -12487.445} C_VEL
LIN {X 0,Y 385.293,Z 514.875,A -85,B 0,C 180,E1 -12487.899,E2 -12487.899} C_VEL
LIN {X 0,Y 384.473,Z 527.353,A -85,B 0,C 180,E1 -12488.484,E2 -12488.484} C_VEL
LIN {X 0,Y 383.412,Z 541.172,A -85,B 0,C 180,E1 -12489.364,E2 -12489.364} C_VEL
LIN {X 0,Y 382.2,Z 553.735,A -85,B 0,C 180,E1 -12490.39,E2 -12490.39} C_VEL
LIN {X 0,Y 380.9,Z 565.449,A -85,B 0,C 180,E1 -12491.579,E2 -12491.579} C_VEL
LIN {X 0,Y 379.743,Z 575.19,A -85,B 0,C 180,E1 -12492.774,E2 -12492.774} C_VEL
LIN {X 0,Y 378.368,Z 585.954,A -85,B 0,C 180,E1 -12494.374,E2 -12494.374} C_VEL
LIN {X 0,Y 377.397,Z 594.837,A -85,B 0,C 180,E1 -12495.989,E2 -12495.989} C_VEL
LIN {X 0,Y 376.343,Z 603.342,A -85,B 0,C 180,E1 -12497.871,E2 -12497.871} C_VEL
LIN {X 0,Y 375.602,Z 610.195,A -85,B 0,C 180,E1 -12499.759,E2 -12499.759} C_VEL
LIN {X 0,Y 375.123,Z 614.925,A -85,B 0,C 180,E1 -12501.378,E2 -12501.378} C_VEL
LIN {X 0,Y 374.784,Z 619.819,A -85,B 0,C 180,E1 -12503.538,E2 -12503.538} C_VEL
LIN {X 0,Y 374.725,Z 620.6,A -85,B 0,C 180,E1 -12503.975,E2 -12503.975} C_VEL
LIN {X 0,Y 373.95,Z 622.096,A -85,B 0,C 180,E1 -12504.845,E2 -12504.845} C_VEL
LIN {X 0,Y 370.944,Z 623.96,A -85,B 0,C 180,E1 -12506.269,E2 -12506.269} C_VEL
LIN {X 0,Y 368.462,Z 625.037,A -85,B 0,C 180,E1 -12507.432,E2 -12507.432} C_VEL
LIN {X 0,Y 367.42,Z 625.592,A -85,B 0,C 180,E1 -12508.339,E2 -12508.339} C_VEL
LIN {X 0,Y 367.346,Z 625.719,A -85,B 0,C 180,E1 -12508.646,E2 -12508.646} C_VEL
LIN {X 0,Y 367.373,Z 626.022,A -85,B 0,C 180,E1 -12509.998,E2 -12509.998} C_VEL
LIN {X 0,Y 367.357,Z 625.397,A -85,B 0,C 180,E1 -12512.191,E2 -12512.191} C_VEL
LIN {X 0,Y 367.507,Z 623.436,A -85,B 0,C 180,E1 -12514.385,E2 -12514.385} C_VEL
LIN {X 0,Y 367.648,Z 620.09,A -85,B 0,C 180,E1 -12516.584,E2 -12516.584} C_VEL
LIN {X 0,Y 368.065,Z 615.259,A -85,B 0,C 180,E1 -12518.785,E2 -12518.785} C_VEL
LIN {X 0,Y 368.734,Z 608.797,A -85,B 0,C 180,E1 -12520.986,E2 -12520.986} C_VEL
LIN {X 0,Y 369.652,Z 601.602,A -85,B 0,C 180,E1 -12522.907,E2 -12522.907} C_VEL
LIN {X 0,Y 370.622,Z 593.157,A -85,B 0,C 180,E1 -12524.738,E2 -12524.738} C_VEL
LIN {X 0,Y 371.89,Z 583.348,A -85,B 0,C 180,E1 -12526.466,E2 -12526.466} C_VEL
LIN {X 0,Y 373.278,Z 572.987,A -85,B 0,C 180,E1 -12527.955,E2 -12527.955} C_VEL
LIN {X 0,Y 374.647,Z 561.559,A -85,B 0,C 180,E1 -12529.305,E2 -12529.305} C_VEL
LIN {X 0,Y 376.069,Z 548.889,A -85,B 0,C 180,E1 -12530.51,E2 -12530.51} C_VEL
LIN {X 0,Y 377.157,Z 536.479,A -85,B 0,C 180,E1 -12531.454,E2 -12531.454} C_VEL
LIN {X 0,Y 378.202,Z 522.887,A -85,B 0,C 180,E1 -12532.246,E2 -12532.246} C_VEL
LIN {X 0,Y 379.079,Z 508.662,A -85,B 0,C 180,E1 -12532.839,E2 -12532.839} C_VEL
LIN {X 0,Y 379.659,Z 495.029,A -85,B 0,C 180,E1 -12533.198,E2 -12533.198} C_VEL
LIN {X 0,Y 381.55,Z 396.363,A -85,B 0,C 180,E1 -12535.072,E2 -12535.072} C_VEL
LIN {X 0,Y 377.304,Z 375.93,A -85,B 0,C 180,E1 -12535.797,E2 -12535.797} C_VEL
LIN {X 0,Y 372.505,Z 363.995,A -85,B 0,C 180,E1 -12536.432,E2 -12536.432} C_VEL
LIN {X 0,Y 369.761,Z 351.708,A -85,B 0,C 180,E1 -12539.613,E2 -12539.613} C_VEL
LIN {X 0,Y 368.932,Z 348.161,A -85,B 0,C 180,E1 -12540.594,E2 -12540.594} C_VEL
LIN {X 0,Y 368.89,Z 348.163,A -85,B 0,C 180,E1 -12543.536,E2 -12543.536} C_VEL
LIN {X 0,Y 368.892,Z 348.163,A -85,B 0,C 180,E1 -12546.853,E2 -12546.853} C_VEL
LIN {X 0,Y 368.875,Z 348.162,A -85,B 0,C 180,E1 -12550.372,E2 -12550.372} C_VEL
LIN {X 0,Y 368.869,Z 348.16,A -85,B 0,C 180,E1 -12553.613,E2 -12553.613} C_VEL
LIN {X 0,Y 368.875,Z 348.161,A -85,B 0,C 180,E1 -12556.694,E2 -12556.694} C_VEL
LIN {X 0,Y 368.873,Z 348.16,A -85,B 0,C 180,E1 -12559.647,E2 -12559.647} C_VEL
LIN {X 0,Y 368.887,Z 348.156,A -85,B 0,C 180,E1 -12563.144,E2 -12563.144} C_VEL
LIN {X 0,Y 368.884,Z 348.151,A -85,B 0,C 180,E1 -12566.46,E2 -12566.46} C_VEL
LIN {X 0,Y 368.883,Z 348.158,A -85,B 0,C 180,E1 -12569.042,E2 -12569.042} C_VEL
LIN {X 0,Y 368.894,Z 348.153,A -85,B 0,C 180,E1 -12571.557,E2 -12571.557} C_VEL
LIN {X 0,Y 368.9,Z 348.153,A -85,B 0,C 180,E1 -12575.22,E2 -12575.22} C_VEL
LIN {X 0,Y 368.896,Z 348.151,A -85,B 0,C 180,E1 -12578.778,E2 -12578.778} C_VEL
LIN {X 0,Y 368.977,Z 348.134,A -85,B 0,C 180,E1 -12582.256,E2 -12582.256} C_VEL
LIN {X 0,Y 369.023,Z 348.141,A -85,B 0,C 180,E1 -12586.227,E2 -12586.227} C_VEL
LIN {X 0,Y 369.048,Z 348.138,A -85,B 0,C 180,E1 -12590.131,E2 -12590.131} C_VEL
LIN {X 0,Y 369.137,Z 348.126,A -85,B 0,C 180,E1 -12593.44,E2 -12593.44} C_VEL
LIN {X 0,Y 369.29,Z 348.108,A -85,B 0,C 180,E1 -12597.819,E2 -12597.819} C_VEL
LIN {X 0,Y 369.287,Z 348.11,A -85,B 0,C 180,E1 -12602.181,E2 -12602.181} C_VEL
LIN {X 0,Y 369.145,Z 348.13,A -85,B 0,C 180,E1 -12606.559,E2 -12606.559} C_VEL
LIN {X 0,Y 369.042,Z 348.137,A -85,B 0,C 180,E1 -12609.869,E2 -12609.869} C_VEL
LIN {X 0,Y 369.023,Z 348.138,A -85,B 0,C 180,E1 -12613.772,E2 -12613.772} C_VEL
LIN {X 0,Y 368.977,Z 348.144,A -85,B 0,C 180,E1 -12617.743,E2 -12617.743} C_VEL
LIN {X 0,Y 368.895,Z 348.145,A -85,B 0,C 180,E1 -12621.222,E2 -12621.222} C_VEL
LIN {X 0,Y 368.894,Z 348.148,A -85,B 0,C 180,E1 -12623.875,E2 -12623.875} C_VEL
LIN {X 0,Y 368.845,Z 348.159,A -85,B 0,C 180,E1 -12627.213,E2 -12627.213} C_VEL
LIN {X 0,Y 368.88,Z 348.147,A -85,B 0,C 180,E1 -12629.693,E2 -12629.693} C_VEL
LIN {X 0,Y 368.883,Z 348.155,A -85,B 0,C 180,E1 -12633.044,E2 -12633.044} C_VEL
LIN {X 0,Y 368.898,Z 348.158,A -85,B 0,C 180,E1 -12636.199,E2 -12636.199} C_VEL
LIN {X 0,Y 368.861,Z 348.162,A -85,B 0,C 180,E1 -12638.958,E2 -12638.958} C_VEL
LIN {X 0,Y 368.846,Z 348.165,A -85,B 0,C 180,E1 -12642.007,E2 -12642.007} C_VEL
LIN {X 0,Y 368.862,Z 348.162,A -85,B 0,C 180,E1 -12645.176,E2 -12645.176} C_VEL
LIN {X 0,Y 368.85,Z 348.169,A -85,B 0,C 180,E1 -12648.176,E2 -12648.176} C_VEL
LIN {X 0,Y 368.865,Z 348.164,A -85,B 0,C 180,E1 -12651.368,E2 -12651.368} C_VEL
LIN {X 0,Y 368.922,Z 348.157,A -85,B 0,C 180,E1 -12655.147,E2 -12655.147} C_VEL
LIN {X 0,Y 368.933,Z 348.276,A -85,B 0,C 180,E1 -12658.243,E2 -12658.243} C_VEL
LIN {X 0,Y 371.934,Z 361.067,A -85,B 0,C 180,E1 -12661.505,E2 -12661.505} C_VEL
LIN {X 0,Y 373.866,Z 370.329,A -85,B 0,C 180,E1 -12663.742,E2 -12663.742} C_VEL
LIN {X 0,Y 375.63,Z 375.549,A -85,B 0,C 180,E1 -12663.983,E2 -12663.983} C_VEL
LIN {X 0,Y 380.643,Z 400.196,A -85,B 0,C 180,E1 -12664.854,E2 -12664.854} C_VEL
LIN {X 0,Y 381.422,Z 405.287,A -85,B 0,C 180,E1 -12665.012,E2 -12665.012} C_VEL
LIN {X 0,Y 379.349,Z 507.26,A -85,B 0,C 180,E1 -12666.962,E2 -12666.962} C_VEL
LIN {X 0,Y 378.555,Z 522.095,A -85,B 0,C 180,E1 -12667.452,E2 -12667.452} C_VEL
LIN {X 0,Y 377.574,Z 536.144,A -85,B 0,C 180,E1 -12668.146,E2 -12668.146} C_VEL
LIN {X 0,Y 376.469,Z 548.696,A -85,B 0,C 180,E1 -12668.973,E2 -12668.973} C_VEL
LIN {X 0,Y 375.248,Z 561.098,A -85,B 0,C 180,E1 -12670.015,E2 -12670.015} C_VEL
LIN {X 0,Y 373.856,Z 572.726,A -85,B 0,C 180,E1 -12671.222,E2 -12671.222} C_VEL
LIN {X 0,Y 372.596,Z 582.406,A -85,B 0,C 180,E1 -12672.436,E2 -12672.436} C_VEL
LIN {X 0,Y 371.196,Z 593.135,A -85,B 0,C 180,E1 -12674.068,E2 -12674.068} C_VEL
LIN {X 0,Y 370.164,Z 601.993,A -85,B 0,C 180,E1 -12675.712,E2 -12675.712} C_VEL
LIN {X 0,Y 369.193,Z 610.484,A -85,B 0,C 180,E1 -12677.636,E2 -12677.636} C_VEL
LIN {X 0,Y 368.357,Z 617.321,A -85,B 0,C 180,E1 -12679.559,E2 -12679.559} C_VEL
LIN {X 0,Y 367.915,Z 622.034,A -85,B 0,C 180,E1 -12681.212,E2 -12681.212} C_VEL
LIN {X 0,Y 367.562,Z 626.923,A -85,B 0,C 180,E1 -12683.414,E2 -12683.414} C_VEL
LIN {X 0,Y 367.425,Z 630.32,A -85,B 0,C 180,E1 -12685.614,E2 -12685.614} C_VEL
LIN {X 0,Y 367.313,Z 632.324,A -85,B 0,C 180,E1 -12687.809,E2 -12687.809} C_VEL
LIN {X 0,Y 367.372,Z 632.985,A -85,B 0,C 180,E1 -12690.002,E2 -12690.002} C_VEL
LIN {X 0,Y 367.314,Z 632.313,A -85,B 0,C 180,E1 -12692.195,E2 -12692.195} C_VEL
LIN {X 0,Y 367.425,Z 630.298,A -85,B 0,C 180,E1 -12694.39,E2 -12694.39} C_VEL
LIN {X 0,Y 367.589,Z 626.895,A -85,B 0,C 180,E1 -12696.589,E2 -12696.589} C_VEL
LIN {X 0,Y 367.918,Z 622.001,A -85,B 0,C 180,E1 -12698.792,E2 -12698.792} C_VEL
LIN {X 0,Y 368.514,Z 615.464,A -85,B 0,C 180,E1 -12700.996,E2 -12700.996} C_VEL
LIN {X 0,Y 369.485,Z 608.191,A -85,B 0,C 180,E1 -12702.916,E2 -12702.916} C_VEL
LIN {X 0,Y 370.452,Z 599.185,A -85,B 0,C 180,E1 -12704.841,E2 -12704.841} C_VEL
LIN {X 0,Y 371.668,Z 589.727,A -85,B 0,C 180,E1 -12706.479,E2 -12706.479} C_VEL
LIN {X 0,Y 373.031,Z 579.263,A -85,B 0,C 180,E1 -12707.971,E2 -12707.971} C_VEL
LIN {X 0,Y 374.422,Z 567.71,A -85,B 0,C 180,E1 -12709.32,E2 -12709.32} C_VEL
LIN {X 0,Y 375.905,Z 554.891,A -85,B 0,C 180,E1 -12710.523,E2 -12710.523} C_VEL
LIN {X 0,Y 377.076,Z 541.853,A -85,B 0,C 180,E1 -12711.494,E2 -12711.494} C_VEL
LIN {X 0,Y 378.113,Z 528.433,A -85,B 0,C 180,E1 -12712.255,E2 -12712.255} C_VEL
LIN {X 0,Y 378.982,Z 514.658,A -85,B 0,C 180,E1 -12712.813,E2 -12712.813} C_VEL
LIN {X 0,Y 379.511,Z 500.541,A -85,B 0,C 180,E1 -12713.175,E2 -12713.175} C_VEL
LIN {X 0,Y 381.424,Z 405.637,A -85,B 0,C 180,E1 -12714.968,E2 -12714.968} C_VEL
LIN {X 0,Y 377.34,Z 383.553,A -85,B 0,C 180,E1 -12715.711,E2 -12715.711} C_VEL
LIN {X 0,Y 374.968,Z 373.193,A -85,B 0,C 180,E1 -12716.101,E2 -12716.101} C_VEL
LIN {X 0,Y 374.545,Z 372.122,A -85,B 0,C 180,E1 -12716.196,E2 -12716.196} C_VEL
LIN {X 0,Y 373.395,Z 368.043,A -85,B 0,C 180,E1 -12716.775,E2 -12716.775} C_VEL
LIN {X 0,Y 370.729,Z 355.611,A -85,B 0,C 180,E1 -12719.845,E2 -12719.845} C_VEL
LIN {X 0,Y 368.915,Z 348.157,A -85,B 0,C 180,E1 -12721.799,E2 -12721.799} C_VEL
LIN {X 0,Y 368.934,Z 348.152,A -85,B 0,C 180,E1 -12725.002,E2 -12725.002} C_VEL
LIN {X 0,Y 368.912,Z 348.152,A -85,B 0,C 180,E1 -12728.641,E2 -12728.641} C_VEL
LIN {X 0,Y 368.886,Z 348.157,A -85,B 0,C 180,E1 -12732.01,E2 -12732.01} C_VEL
LIN {X 0,Y 368.885,Z 348.162,A -85,B 0,C 180,E1 -12735.177,E2 -12735.177} C_VEL
LIN {X 0,Y 368.888,Z 348.157,A -85,B 0,C 180,E1 -12738.178,E2 -12738.178} C_VEL
LIN {X 0,Y 368.914,Z 348.156,A -85,B 0,C 180,E1 -12741.36,E2 -12741.36} C_VEL
LIN {X 0,Y 368.942,Z 348.152,A -85,B 0,C 180,E1 -12745.147,E2 -12745.147} C_VEL
LIN {X 0,Y 368.945,Z 348.276,A -85,B 0,C 180,E1 -12747.179,E2 -12747.179} C_VEL
LIN {X 0,Y 372.552,Z 358.013,A -85,B 0,C 180,E1 -12750.202,E2 -12750.202} C_VEL
LIN {X 0,Y 375.421,Z 367.77,A -85,B 0,C 180,E1 -12752.832,E2 -12752.832} C_VEL
LIN {X 0,Y 376.997,Z 374.974,A -85,B 0,C 180,E1 -12754.611,E2 -12754.611} C_VEL
LIN {X 0,Y 377.287,Z 379.029,A -85,B 0,C 180,E1 -12755.514,E2 -12755.514} C_VEL
LIN {X 0,Y 377.011,Z 383.319,A -85,B 0,C 180,E1 -12756.355,E2 -12756.355} C_VEL
LIN {X 0,Y 380.466,Z 396.663,A -85,B 0,C 180,E1 -12757.253,E2 -12757.253} C_VEL
LIN {X 0,Y 382.126,Z 404.8,A -85,B 0,C 180,E1 -12757.721,E2 -12757.721} C_VEL
LIN {X 0,Y 378.288,Z 481.612,A -85,B 0,C 180,E1 -12759.933,E2 -12759.933} C_VEL
LIN {X 0,Y 377.561,Z 496.786,A -85,B 0,C 180,E1 -12760.424,E2 -12760.424} C_VEL
LIN {X 0,Y 376.759,Z 510.304,A -85,B 0,C 180,E1 -12761.088,E2 -12761.088} C_VEL
LIN {X 0,Y 375.84,Z 522.211,A -85,B 0,C 180,E1 -12761.888,E2 -12761.888} C_VEL
LIN {X 0,Y 374.807,Z 533.48,A -85,B 0,C 180,E1 -12762.851,E2 -12762.851} C_VEL
LIN {X 0,Y 373.812,Z 542.789,A -85,B 0,C 180,E1 -12763.825,E2 -12763.825} C_VEL
LIN {X 0,Y 372.769,Z 551.869,A -85,B 0,C 180,E1 -12764.975,E2 -12764.975} C_VEL
LIN {X 0,Y 371.664,Z 560.649,A -85,B 0,C 180,E1 -12766.328,E2 -12766.328} C_VEL
LIN {X 0,Y 370.573,Z 569.258,A -85,B 0,C 180,E1 -12767.959,E2 -12767.959} C_VEL
LIN {X 0,Y 369.726,Z 576.128,A -85,B 0,C 180,E1 -12769.596,E2 -12769.596} C_VEL
LIN {X 0,Y 369.003,Z 581.602,A -85,B 0,C 180,E1 -12771.236,E2 -12771.236} C_VEL
LIN {X 0,Y 368.596,Z 585.046,A -85,B 0,C 180,E1 -12772.524,E2 -12772.524} C_VEL
LIN {X 0,Y 367.957,Z 588.98,A -85,B 0,C 180,E1 -12774.52,E2 -12774.52} C_VEL
LIN {X 0,Y 367.947,Z 590.492,A -85,B 0,C 180,E1 -12775.618,E2 -12775.618} C_VEL
LIN {X 0,Y 367.855,Z 591.549,A -85,B 0,C 180,E1 -12776.714,E2 -12776.714} C_VEL
LIN {X 0,Y 367.7,Z 592.168,A -85,B 0,C 180,E1 -12777.809,E2 -12777.809} C_VEL
LIN {X 0,Y 367.589,Z 592.376,A -85,B 0,C 180,E1 -12778.905,E2 -12778.905} C_VEL
LIN {X 0,Y 367.545,Z 592.139,A -85,B 0,C 180,E1 -12780,E2 -12780} C_VEL
LIN {X 0,Y 367.551,Z 591.441,A -85,B 0,C 180,E1 -12781.096,E2 -12781.096} C_VEL
LIN {X 0,Y 367.56,Z 590.331,A -85,B 0,C 180,E1 -12782.192,E2 -12782.192} C_VEL
LIN {X 0,Y 367.597,Z 587.812,A -85,B 0,C 180,E1 -12783.837,E2 -12783.837} C_VEL
LIN {X 0,Y 367.772,Z 584.229,A -85,B 0,C 180,E1 -12785.483,E2 -12785.483} C_VEL
LIN {X 0,Y 367.991,Z 579.48,A -85,B 0,C 180,E1 -12787.131,E2 -12787.131} C_VEL
LIN {X 0,Y 368.293,Z 573.387,A -85,B 0,C 180,E1 -12788.781,E2 -12788.781} C_VEL
LIN {X 0,Y 368.814,Z 565.777,A -85,B 0,C 180,E1 -12790.43,E2 -12790.43} C_VEL
LIN {X 0,Y 369.283,Z 558.011,A -85,B 0,C 180,E1 -12791.806,E2 -12791.806} C_VEL
LIN {X 0,Y 370.101,Z 547.513,A -85,B 0,C 180,E1 -12793.312,E2 -12793.312} C_VEL
LIN {X 0,Y 370.732,Z 537.573,A -85,B 0,C 180,E1 -12794.474,E2 -12794.474} C_VEL
LIN {X 0,Y 371.3,Z 526.728,A -85,B 0,C 180,E1 -12795.507,E2 -12795.507} C_VEL
LIN {X 0,Y 371.993,Z 513.839,A -85,B 0,C 180,E1 -12796.463,E2 -12796.463} C_VEL
LIN {X 0,Y 372.537,Z 500.983,A -85,B 0,C 180,E1 -12797.179,E2 -12797.179} C_VEL
LIN {X 0,Y 373.027,Z 486.659,A -85,B 0,C 180,E1 -12797.722,E2 -12797.722} C_VEL
LIN {X 0,Y 374.951,Z 400.607,A -85,B 0,C 180,E1 -12799.862,E2 -12799.862} C_VEL
LIN {X 0,Y 371.584,Z 378.823,A -85,B 0,C 180,E1 -12800.583,E2 -12800.583} C_VEL
LIN {X 0,Y 372.16,Z 365.869,A -85,B 0,C 180,E1 -12803.07,E2 -12803.07} C_VEL
LIN {X 0,Y 371.192,Z 359.225,A -85,B 0,C 180,E1 -12804.42,E2 -12804.42} C_VEL
LIN {X 0,Y 369.02,Z 348.145,A -85,B 0,C 180,E1 -12806.734,E2 -12806.734} C_VEL
LIN {X 0,Y 368.925,Z 348.156,A -85,B 0,C 180,E1 -12809.69,E2 -12809.69} C_VEL
LIN {X 0,Y 368.903,Z 348.156,A -85,B 0,C 180,E1 -12813.043,E2 -12813.043} C_VEL
LIN {X 0,Y 368.922,Z 348.155,A -85,B 0,C 180,E1 -12816.196,E2 -12816.196} C_VEL
LIN {X 0,Y 368.88,Z 348.158,A -85,B 0,C 180,E1 -12818.956,E2 -12818.956} C_VEL
LIN {X 0,Y 368.877,Z 348.164,A -85,B 0,C 180,E1 -12822.007,E2 -12822.007} C_VEL
LIN {X 0,Y 368.884,Z 348.16,A -85,B 0,C 180,E1 -12825.175,E2 -12825.175} C_VEL
LIN {X 0,Y 368.875,Z 348.161,A -85,B 0,C 180,E1 -12828.175,E2 -12828.175} C_VEL
LIN {X 0,Y 368.881,Z 348.163,A -85,B 0,C 180,E1 -12831.365,E2 -12831.365} C_VEL
LIN {X 0,Y 368.936,Z 348.15,A -85,B 0,C 180,E1 -12835.145,E2 -12835.145} C_VEL
LIN {X 0,Y 368.901,Z 348.158,A -85,B 0,C 180,E1 -12839.042,E2 -12839.042} C_VEL
LIN {X 0,Y 368.95,Z 348.232,A -85,B 0,C 180,E1 -12839.563,E2 -12839.563} C_VEL
LIN {X 0,Y 371.667,Z 360.234,A -85,B 0,C 180,E1 -12842.716,E2 -12842.716} C_VEL
LIN {X 0,Y 372.55,Z 364.214,A -85,B 0,C 180,E1 -12843.706,E2 -12843.706} C_VEL
LIN {X 0,Y 377.845,Z 377.799,A -85,B 0,C 180,E1 -12844.385,E2 -12844.385} C_VEL
LIN {X 0,Y 381.559,Z 396.633,A -85,B 0,C 180,E1 -12845.037,E2 -12845.037} C_VEL
LIN {X 0,Y 379.422,Z 501.041,A -85,B 0,C 180,E1 -12847.035,E2 -12847.035} C_VEL
LIN {X 0,Y 378.725,Z 514.953,A -85,B 0,C 180,E1 -12847.495,E2 -12847.495} C_VEL
LIN {X 0,Y 377.876,Z 527.428,A -85,B 0,C 180,E1 -12848.089,E2 -12848.089} C_VEL
LIN {X 0,Y 376.795,Z 540.547,A -85,B 0,C 180,E1 -12848.928,E2 -12848.928} C_VEL
LIN {X 0,Y 375.667,Z 552.383,A -85,B 0,C 180,E1 -12849.892,E2 -12849.892} C_VEL
LIN {X 0,Y 374.334,Z 564.348,A -85,B 0,C 180,E1 -12851.102,E2 -12851.102} C_VEL
LIN {X 0,Y 372.937,Z 575.261,A -85,B 0,C 180,E1 -12852.45,E2 -12852.45} C_VEL
LIN {X 0,Y 371.738,Z 584.401,A -85,B 0,C 180,E1 -12853.806,E2 -12853.806} C_VEL
LIN {X 0,Y 370.559,Z 593.701,A -85,B 0,C 180,E1 -12855.474,E2 -12855.474} C_VEL
LIN {X 0,Y 369.698,Z 601.185,A -85,B 0,C 180,E1 -12857.092,E2 -12857.092} C_VEL
LIN {X 0,Y 368.772,Z 608.46,A -85,B 0,C 180,E1 -12859.012,E2 -12859.012} C_VEL
LIN {X 0,Y 368.24,Z 613.551,A -85,B 0,C 180,E1 -12860.662,E2 -12860.662} C_VEL
LIN {X 0,Y 367.775,Z 618.827,A -85,B 0,C 180,E1 -12862.863,E2 -12862.863} C_VEL
LIN {X 0,Y 367.576,Z 621.77,A -85,B 0,C 180,E1 -12864.513,E2 -12864.513} C_VEL
LIN {X 0,Y 367.388,Z 624.479,A -85,B 0,C 180,E1 -12866.708,E2 -12866.708} C_VEL
LIN {X 0,Y 367.346,Z 625.719,A -85,B 0,C 180,E1 -12868.646,E2 -12868.646} C_VEL
LIN {X 0,Y 366.696,Z 626.036,A -85,B 0,C 180,E1 -12869.56,E2 -12869.56} C_VEL
LIN {X 0,Y 363.824,Z 626.04,A -85,B 0,C 180,E1 -12871.05,E2 -12871.05} C_VEL
LIN {X 0,Y 361.398,Z 625.53,A -85,B 0,C 180,E1 -12872.251,E2 -12872.251} C_VEL
LIN {X 0,Y 360.382,Z 624.819,A -85,B 0,C 180,E1 -12873.176,E2 -12873.176} C_VEL
LIN {X 0,Y 360.314,Z 624.515,A -85,B 0,C 180,E1 -12873.488,E2 -12873.488} C_VEL
LIN {X 0,Y 360.477,Z 622.008,A -85,B 0,C 180,E1 -12875.592,E2 -12875.592} C_VEL
LIN {X 0,Y 360.774,Z 617.935,A -85,B 0,C 180,E1 -12877.836,E2 -12877.836} C_VEL
LIN {X 0,Y 361.342,Z 612.309,A -85,B 0,C 180,E1 -12880.08,E2 -12880.08} C_VEL
LIN {X 0,Y 362.064,Z 605.962,A -85,B 0,C 180,E1 -12882.042,E2 -12882.042} C_VEL
LIN {X 0,Y 363.177,Z 598.066,A -85,B 0,C 180,E1 -12883.996,E2 -12883.996} C_VEL
LIN {X 0,Y 364.209,Z 589.807,A -85,B 0,C 180,E1 -12885.671,E2 -12885.671} C_VEL
LIN {X 0,Y 365.574,Z 579.856,A -85,B 0,C 180,E1 -12887.334,E2 -12887.334} C_VEL
LIN {X 0,Y 367.084,Z 568.776,A -85,B 0,C 180,E1 -12888.847,E2 -12888.847} C_VEL
LIN {X 0,Y 368.463,Z 557.749,A -85,B 0,C 180,E1 -12890.078,E2 -12890.078} C_VEL
LIN {X 0,Y 369.723,Z 545.776,A -85,B 0,C 180,E1 -12891.17,E2 -12891.17} C_VEL
LIN {X 0,Y 370.932,Z 532.648,A -85,B 0,C 180,E1 -12892.111,E2 -12892.111} C_VEL
LIN {X 0,Y 371.985,Z 518.762,A -85,B 0,C 180,E1 -12892.859,E2 -12892.859} C_VEL
LIN {X 0,Y 372.723,Z 505.588,A -85,B 0,C 180,E1 -12893.361,E2 -12893.361} C_VEL
LIN {X 0,Y 373.261,Z 488.052,A -85,B 0,C 180,E1 -12893.767,E2 -12893.767} C_VEL
LIN {X 0,Y 375.078,Z 397.214,A -85,B 0,C 180,E1 -12895.519,E2 -12895.519} C_VEL
LIN {X 0,Y 371.201,Z 378.528,A -85,B 0,C 180,E1 -12896.2,E2 -12896.2} C_VEL
LIN {X 0,Y 365.298,Z 364.092,A -85,B 0,C 180,E1 -12896.989,E2 -12896.989} C_VEL
LIN {X 0,Y 362.773,Z 352.827,A -85,B 0,C 180,E1 -12899.978,E2 -12899.978} C_VEL
LIN {X 0,Y 361.854,Z 349.041,A -85,B 0,C 180,E1 -12901.061,E2 -12901.061} C_VEL
LIN {X 0,Y 361.848,Z 349.041,A -85,B 0,C 180,E1 -12904.279,E2 -12904.279} C_VEL
LIN {X 0,Y 361.852,Z 349.037,A -85,B 0,C 180,E1 -12907.22,E2 -12907.22} C_VEL
LIN {X 0,Y 361.801,Z 349.042,A -85,B 0,C 180,E1 -12910.749,E2 -12910.749} C_VEL
LIN {X 0,Y 361.803,Z 349.041,A -85,B 0,C 180,E1 -12914.368,E2 -12914.368} C_VEL
LIN {X 0,Y 361.82,Z 349.039,A -85,B 0,C 180,E1 -12917.568,E2 -12917.568} C_VEL
LIN {X 0,Y 361.832,Z 349.027,A -85,B 0,C 180,E1 -12921.571,E2 -12921.571} C_VEL
LIN {X 0,Y 361.862,Z 349.037,A -85,B 0,C 180,E1 -12924.654,E2 -12924.654} C_VEL
LIN {X 0,Y 361.822,Z 349.028,A -85,B 0,C 180,E1 -12928.369,E2 -12928.369} C_VEL
LIN {X 0,Y 361.854,Z 349.034,A -85,B 0,C 180,E1 -12930.951,E2 -12930.951} C_VEL
LIN {X 0,Y 361.86,Z 349.021,A -85,B 0,C 180,E1 -12934.705,E2 -12934.705} C_VEL
LIN {X 0,Y 361.841,Z 349.036,A -85,B 0,C 180,E1 -12938.344,E2 -12938.344} C_VEL
LIN {X 0,Y 361.907,Z 349.014,A -85,B 0,C 180,E1 -12942.084,E2 -12942.084} C_VEL
LIN {X 0,Y 361.947,Z 349.021,A -85,B 0,C 180,E1 -12945.379,E2 -12945.379} C_VEL
LIN {X 0,Y 361.955,Z 349.025,A -85,B 0,C 180,E1 -12948.804,E2 -12948.804} C_VEL
LIN {X 0,Y 362.061,Z 349.006,A -85,B 0,C 180,E1 -12952.191,E2 -12952.191} C_VEL
LIN {X 0,Y 362.072,Z 349.008,A -85,B 0,C 180,E1 -12954.43,E2 -12954.43} C_VEL
LIN {X 0,Y 362.253,Z 348.984,A -85,B 0,C 180,E1 -12957.776,E2 -12957.776} C_VEL
LIN {X 0,Y 362.25,Z 348.987,A -85,B 0,C 180,E1 -12962.224,E2 -12962.224} C_VEL
LIN {X 0,Y 362.108,Z 349.005,A -85,B 0,C 180,E1 -12966.687,E2 -12966.687} C_VEL
LIN {X 0,Y 361.979,Z 349.018,A -85,B 0,C 180,E1 -12970.063,E2 -12970.063} C_VEL
LIN {X 0,Y 361.984,Z 349.015,A -85,B 0,C 180,E1 -12973.899,E2 -12973.899} C_VEL
LIN {X 0,Y 361.914,Z 349.024,A -85,B 0,C 180,E1 -12976.935,E2 -12976.935} C_VEL
LIN {X 0,Y 361.87,Z 349.026,A -85,B 0,C 180,E1 -12980.462,E2 -12980.462} C_VEL
LIN {X 0,Y 361.847,Z 349.028,A -85,B 0,C 180,E1 -12984.102,E2 -12984.102} C_VEL
LIN {X 0,Y 361.822,Z 349.033,A -85,B 0,C 180,E1 -12987.786,E2 -12987.786} C_VEL
LIN {X 0,Y 361.832,Z 349.036,A -85,B 0,C 180,E1 -12991.286,E2 -12991.286} C_VEL
LIN {X 0,Y 361.838,Z 349.039,A -85,B 0,C 180,E1 -12994.282,E2 -12994.282} C_VEL
LIN {X 0,Y 361.845,Z 349.036,A -85,B 0,C 180,E1 -12997.223,E2 -12997.223} C_VEL
LIN {X 0,Y 361.798,Z 349.041,A -85,B 0,C 180,E1 -13000.752,E2 -13000.752} C_VEL
LIN {X 0,Y 361.8,Z 349.046,A -85,B 0,C 180,E1 -13004.371,E2 -13004.371} C_VEL
LIN {X 0,Y 361.812,Z 349.042,A -85,B 0,C 180,E1 -13007.572,E2 -13007.572} C_VEL
LIN {X 0,Y 361.832,Z 349.041,A -85,B 0,C 180,E1 -13011.573,E2 -13011.573} C_VEL
LIN {X 0,Y 361.862,Z 349.038,A -85,B 0,C 180,E1 -13014.658,E2 -13014.658} C_VEL
LIN {X 0,Y 361.874,Z 349.08,A -85,B 0,C 180,E1 -13017.762,E2 -13017.762} C_VEL
LIN {X 0,Y 364.607,Z 360.499,A -85,B 0,C 180,E1 -13020.76,E2 -13020.76} C_VEL
LIN {X 0,Y 366.667,Z 370.361,A -85,B 0,C 180,E1 -13023.187,E2 -13023.187} C_VEL
LIN {X 0,Y 369.4,Z 377.389,A -85,B 0,C 180,E1 -13023.55,E2 -13023.55} C_VEL
LIN {X 0,Y 374.339,Z 401.984,A -85,B 0,C 180,E1 -13024.438,E2 -13024.438} C_VEL
LIN {X 0,Y 374.965,Z 405.709,A -85,B 0,C 180,E1 -13024.561,E2 -13024.561} C_VEL
LIN {X 0,Y 372.883,Z 505.73,A -85,B 0,C 180,E1 -13026.502,E2 -13026.502} C_VEL
LIN {X 0,Y 372.134,Z 520.473,A -85,B 0,C 180,E1 -13026.967,E2 -13026.967} C_VEL
LIN {X 0,Y 371.158,Z 533.814,A -85,B 0,C 180,E1 -13027.602,E2 -13027.602} C_VEL
LIN {X 0,Y 369.962,Z 547.524,A -85,B 0,C 180,E1 -13028.493,E2 -13028.493} C_VEL
LIN {X 0,Y 368.698,Z 559.695,A -85,B 0,C 180,E1 -13029.508,E2 -13029.508} C_VEL
LIN {X 0,Y 367.299,Z 571.488,A -85,B 0,C 180,E1 -13030.729,E2 -13030.729} C_VEL
LIN {X 0,Y 365.811,Z 582.342,A -85,B 0,C 180,E1 -13032.1,E2 -13032.1} C_VEL
LIN {X 0,Y 364.351,Z 593.07,A -85,B 0,C 180,E1 -13033.76,E2 -13033.76} C_VEL
LIN {X 0,Y 363.213,Z 601.927,A -85,B 0,C 180,E1 -13035.433,E2 -13035.433} C_VEL
LIN {X 0,Y 362.211,Z 610.418,A -85,B 0,C 180,E1 -13037.394,E2 -13037.394} C_VEL
LIN {X 0,Y 361.322,Z 617.254,A -85,B 0,C 180,E1 -13039.353,E2 -13039.353} C_VEL
LIN {X 0,Y 360.863,Z 621.968,A -85,B 0,C 180,E1 -13041.038,E2 -13041.038} C_VEL
LIN {X 0,Y 360.496,Z 626.857,A -85,B 0,C 180,E1 -13043.284,E2 -13043.284} C_VEL
LIN {X 0,Y 360.338,Z 630.253,A -85,B 0,C 180,E1 -13045.527,E2 -13045.527} C_VEL
LIN {X 0,Y 360.22,Z 632.257,A -85,B 0,C 180,E1 -13047.765,E2 -13047.765} C_VEL
LIN {X 0,Y 360.273,Z 632.918,A -85,B 0,C 180,E1 -13050.002,E2 -13050.002} C_VEL
LIN {X 0,Y 360.221,Z 632.245,A -85,B 0,C 180,E1 -13052.238,E2 -13052.238} C_VEL
LIN {X 0,Y 360.339,Z 630.23,A -85,B 0,C 180,E1 -13054.476,E2 -13054.476} C_VEL
LIN {X 0,Y 360.511,Z 626.826,A -85,B 0,C 180,E1 -13056.719,E2 -13056.719} C_VEL
LIN {X 0,Y 360.866,Z 621.932,A -85,B 0,C 180,E1 -13058.965,E2 -13058.965} C_VEL
LIN {X 0,Y 361.5,Z 615.395,A -85,B 0,C 180,E1 -13061.212,E2 -13061.212} C_VEL
LIN {X 0,Y 362.521,Z 608.121,A -85,B 0,C 180,E1 -13063.169,E2 -13063.169} C_VEL
LIN {X 0,Y 363.554,Z 599.115,A -85,B 0,C 180,E1 -13065.129,E2 -13065.129} C_VEL
LIN {X 0,Y 364.818,Z 589.657,A -85,B 0,C 180,E1 -13066.798,E2 -13066.798} C_VEL
LIN {X 0,Y 366.246,Z 579.192,A -85,B 0,C 180,E1 -13068.316,E2 -13068.316} C_VEL
LIN {X 0,Y 367.71,Z 567.639,A -85,B 0,C 180,E1 -13069.687,E2 -13069.687} C_VEL
LIN {X 0,Y 369.246,Z 554.819,A -85,B 0,C 180,E1 -13070.91,E2 -13070.91} C_VEL
LIN {X 0,Y 370.408,Z 542.307,A -85,B 0,C 180,E1 -13071.862,E2 -13071.862} C_VEL
LIN {X 0,Y 371.445,Z 529.659,A -85,B 0,C 180,E1 -13072.603,E2 -13072.603} C_VEL
LIN {X 0,Y 372.41,Z 515.496,A -85,B 0,C 180,E1 -13073.202,E2 -13073.202} C_VEL
LIN {X 0,Y 372.955,Z 502.024,A -85,B 0,C 180,E1 -13073.57,E2 -13073.57} C_VEL
LIN {X 0,Y 374.972,Z 406.433,A -85,B 0,C 180,E1 -13075.409,E2 -13075.409} C_VEL
LIN {X 0,Y 370.586,Z 383.002,A -85,B 0,C 180,E1 -13076.225,E2 -13076.225} C_VEL
LIN {X 0,Y 369.557,Z 377.863,A -85,B 0,C 180,E1 -13076.434,E2 -13076.434} C_VEL
LIN {X 0,Y 368.99,Z 374.861,A -85,B 0,C 180,E1 -13076.796,E2 -13076.796} C_VEL
LIN {X 0,Y 364.924,Z 362.017,A -85,B 0,C 180,E1 -13078.837,E2 -13078.837} C_VEL
LIN {X 0,Y 362.117,Z 350.159,A -85,B 0,C 180,E1 -13081.931,E2 -13081.931} C_VEL
LIN {X 0,Y 361.859,Z 349.037,A -85,B 0,C 180,E1 -13082.285,E2 -13082.285} C_VEL
LIN {X 0,Y 361.873,Z 349.035,A -85,B 0,C 180,E1 -13085.638,E2 -13085.638} C_VEL
LIN {X 0,Y 361.874,Z 349.031,A -85,B 0,C 180,E1 -13089.027,E2 -13089.027} C_VEL
LIN {X 0,Y 361.842,Z 349.036,A -85,B 0,C 180,E1 -13092.83,E2 -13092.83} C_VEL
LIN {X 0,Y 361.823,Z 349.038,A -85,B 0,C 180,E1 -13095.947,E2 -13095.947} C_VEL
LIN {X 0,Y 361.841,Z 349.038,A -85,B 0,C 180,E1 -13099.245,E2 -13099.245} C_VEL
LIN {X 0,Y 361.869,Z 349.035,A -85,B 0,C 180,E1 -13102.778,E2 -13102.778} C_VEL
LIN {X 0,Y 361.896,Z 349.228,A -85,B 0,C 180,E1 -13105.788,E2 -13105.788} C_VEL
LIN {X 0,Y 364.69,Z 356.333,A -85,B 0,C 180,E1 -13108.28,E2 -13108.28} C_VEL
LIN {X 0,Y 367.566,Z 364.699,A -85,B 0,C 180,E1 -13110.838,E2 -13110.838} C_VEL
LIN {X 0,Y 369.927,Z 373.586,A -85,B 0,C 180,E1 -13113.245,E2 -13113.245} C_VEL
LIN {X 0,Y 370.999,Z 379.774,A -85,B 0,C 180,E1 -13114.772,E2 -13114.772} C_VEL
LIN {X 0,Y 370.889,Z 383.833,A -85,B 0,C 180,E1 -13115.618,E2 -13115.618} C_VEL
LIN {X 0,Y 374.703,Z 398.229,A -85,B 0,C 180,E1 -13116.66,E2 -13116.66} C_VEL
LIN {X 0,Y 376.313,Z 406.46,A -85,B 0,C 180,E1 -13117.154,E2 -13117.154} C_VEL
LIN {X 0,Y 372.028,Z 484.54,A -85,B 0,C 180,E1 -13119.472,E2 -13119.472} C_VEL
LIN {X 0,Y 371.215,Z 499.542,A -85,B 0,C 180,E1 -13120.003,E2 -13120.003} C_VEL
LIN {X 0,Y 370.263,Z 513.29,A -85,B 0,C 180,E1 -13120.744,E2 -13120.744} C_VEL
LIN {X 0,Y 369.149,Z 526.265,A -85,B 0,C 180,E1 -13121.692,E2 -13121.692} C_VEL
LIN {X 0,Y 367.752,Z 539.163,A -85,B 0,C 180,E1 -13122.917,E2 -13122.917} C_VEL
LIN {X 0,Y 366.511,Z 549.556,A -85,B 0,C 180,E1 -13124.174,E2 -13124.174} C_VEL
LIN {X 0,Y 365.248,Z 558.656,A -85,B 0,C 180,E1 -13125.514,E2 -13125.514} C_VEL
LIN {X 0,Y 364.281,Z 566.341,A -85,B 0,C 180,E1 -13126.898,E2 -13126.898} C_VEL
LIN {X 0,Y 363.216,Z 573.858,A -85,B 0,C 180,E1 -13128.561,E2 -13128.561} C_VEL
LIN {X 0,Y 362.231,Z 580.778,A -85,B 0,C 180,E1 -13130.508,E2 -13130.508} C_VEL
LIN {X 0,Y 361.596,Z 585.826,A -85,B 0,C 180,E1 -13132.417,E2 -13132.417} C_VEL
LIN {X 0,Y 360.92,Z 589.583,A -85,B 0,C 180,E1 -13134.413,E2 -13134.413} C_VEL
LIN {X 0,Y 360.874,Z 591.037,A -85,B 0,C 180,E1 -13135.532,E2 -13135.532} C_VEL
LIN {X 0,Y 360.788,Z 592.015,A -85,B 0,C 180,E1 -13136.65,E2 -13136.65} C_VEL
LIN {X 0,Y 360.645,Z 592.587,A -85,B 0,C 180,E1 -13137.766,E2 -13137.766} C_VEL
LIN {X 0,Y 360.527,Z 592.744,A -85,B 0,C 180,E1 -13138.883,E2 -13138.883} C_VEL
LIN {X 0,Y 360.463,Z 592.422,A -85,B 0,C 180,E1 -13140,E2 -13140} C_VEL
LIN {X 0,Y 360.455,Z 591.676,A -85,B 0,C 180,E1 -13141.117,E2 -13141.117} C_VEL
LIN {X 0,Y 360.463,Z 590.515,A -85,B 0,C 180,E1 -13142.235,E2 -13142.235} C_VEL
LIN {X 0,Y 360.522,Z 587.896,A -85,B 0,C 180,E1 -13143.912,E2 -13143.912} C_VEL
LIN {X 0,Y 360.682,Z 584.195,A -85,B 0,C 180,E1 -13145.591,E2 -13145.591} C_VEL
LIN {X 0,Y 360.926,Z 579.295,A -85,B 0,C 180,E1 -13147.271,E2 -13147.271} C_VEL
LIN {X 0,Y 361.343,Z 571.907,A -85,B 0,C 180,E1 -13149.234,E2 -13149.234} C_VEL
LIN {X 0,Y 361.893,Z 563.815,A -85,B 0,C 180,E1 -13150.915,E2 -13150.915} C_VEL
LIN {X 0,Y 362.46,Z 555.55,A -85,B 0,C 180,E1 -13152.315,E2 -13152.315} C_VEL
LIN {X 0,Y 363.135,Z 545.512,A -85,B 0,C 180,E1 -13153.715,E2 -13153.715} C_VEL
LIN {X 0,Y 363.844,Z 534.339,A -85,B 0,C 180,E1 -13154.965,E2 -13154.965} C_VEL
LIN {X 0,Y 364.48,Z 523.439,A -85,B 0,C 180,E1 -13155.949,E2 -13155.949} C_VEL
LIN {X 0,Y 365.122,Z 510.544,A -85,B 0,C 180,E1 -13156.854,E2 -13156.854} C_VEL
LIN {X 0,Y 365.725,Z 497.155,A -85,B 0,C 180,E1 -13157.546,E2 -13157.546} C_VEL
LIN {X 0,Y 366.162,Z 482.815,A -85,B 0,C 180,E1 -13158.029,E2 -13158.029} C_VEL
LIN {X 0,Y 368.018,Z 401.366,A -85,B 0,C 180,E1 -13160.105,E2 -13160.105} C_VEL
LIN {X 0,Y 364.655,Z 379.047,A -85,B 0,C 180,E1 -13160.862,E2 -13160.862} C_VEL
LIN {X 0,Y 365.208,Z 366.826,A -85,B 0,C 180,E1 -13163.235,E2 -13163.235} C_VEL
LIN {X 0,Y 363.963,Z 359.089,A -85,B 0,C 180,E1 -13164.828,E2 -13164.828} C_VEL
LIN {X 0,Y 361.964,Z 349.023,A -85,B 0,C 180,E1 -13166.979,E2 -13166.979} C_VEL
LIN {X 0,Y 361.881,Z 349.032,A -85,B 0,C 180,E1 -13170.327,E2 -13170.327} C_VEL
LIN {X 0,Y 361.861,Z 349.036,A -85,B 0,C 180,E1 -13174.28,E2 -13174.28} C_VEL
LIN {X 0,Y 361.866,Z 349.033,A -85,B 0,C 180,E1 -13177.221,E2 -13177.221} C_VEL
LIN {X 0,Y 361.818,Z 349.038,A -85,B 0,C 180,E1 -13180.75,E2 -13180.75} C_VEL
LIN {X 0,Y 361.822,Z 349.04,A -85,B 0,C 180,E1 -13184.368,E2 -13184.368} C_VEL
LIN {X 0,Y 361.835,Z 349.041,A -85,B 0,C 180,E1 -13187.569,E2 -13187.569} C_VEL
LIN {X 0,Y 361.847,Z 349.038,A -85,B 0,C 180,E1 -13191.571,E2 -13191.571} C_VEL
LIN {X 0,Y 361.875,Z 349.032,A -85,B 0,C 180,E1 -13194.655,E2 -13194.655} C_VEL
LIN {X 0,Y 361.842,Z 349.04,A -85,B 0,C 180,E1 -13198.369,E2 -13198.369} C_VEL
LIN {X 0,Y 361.895,Z 349.23,A -85,B 0,C 180,E1 -13199.14,E2 -13199.14} C_VEL
LIN {X 0,Y 364.487,Z 360.265,A -85,B 0,C 180,E1 -13202.121,E2 -13202.121} C_VEL
LIN {X 0,Y 365.338,Z 364.311,A -85,B 0,C 180,E1 -13203.146,E2 -13203.146} C_VEL
LIN {X 0,Y 371.743,Z 380.332,A -85,B 0,C 180,E1 -13203.985,E2 -13203.985} C_VEL
LIN {X 0,Y 375.112,Z 397.81,A -85,B 0,C 180,E1 -13204.6,E2 -13204.6} C_VEL
LIN {X 0,Y 372.904,Z 501.126,A -85,B 0,C 180,E1 -13206.61,E2 -13206.61} C_VEL
LIN {X 0,Y 372.174,Z 515.031,A -85,B 0,C 180,E1 -13207.077,E2 -13207.077} C_VEL
LIN {X 0,Y 371.201,Z 528.634,A -85,B 0,C 180,E1 -13207.748,E2 -13207.748} C_VEL
LIN {X 0,Y 370.065,Z 541.83,A -85,B 0,C 180,E1 -13208.626,E2 -13208.626} C_VEL
LIN {X 0,Y 368.678,Z 555.304,A -85,B 0,C 180,E1 -13209.785,E2 -13209.785} C_VEL
LIN {X 0,Y 367.247,Z 566.765,A -85,B 0,C 180,E1 -13211.013,E2 -13211.013} C_VEL
LIN {X 0,Y 365.924,Z 577.279,A -85,B 0,C 180,E1 -13212.391,E2 -13212.391} C_VEL
LIN {X 0,Y 364.43,Z 587.719,A -85,B 0,C 180,E1 -13214.048,E2 -13214.048} C_VEL
LIN {X 0,Y 363.367,Z 596.329,A -85,B 0,C 180,E1 -13215.722,E2 -13215.722} C_VEL
LIN {X 0,Y 362.278,Z 604.581,A -85,B 0,C 180,E1 -13217.677,E2 -13217.677} C_VEL
LIN {X 0,Y 361.564,Z 610.334,A -85,B 0,C 180,E1 -13219.357,E2 -13219.357} C_VEL
LIN {X 0,Y 361.043,Z 615.063,A -85,B 0,C 180,E1 -13221.039,E2 -13221.039} C_VEL
LIN {X 0,Y 360.657,Z 619.956,A -85,B 0,C 180,E1 -13223.284,E2 -13223.284} C_VEL
LIN {X 0,Y 360.422,Z 623.364,A -85,B 0,C 180,E1 -13225.525,E2 -13225.525} C_VEL
LIN {X 0,Y 360.264,Z 625.392,A -85,B 0,C 180,E1 -13227.762,E2 -13227.762} C_VEL
LIN {X 0,Y 360.274,Z 626.089,A -85,B 0,C 180,E1 -13229.998,E2 -13229.998} C_VEL
LIN {X 0,Y 360.262,Z 625.464,A -85,B 0,C 180,E1 -13232.234,E2 -13232.234} C_VEL
LIN {X 0,Y 360.314,Z 624.515,A -85,B 0,C 180,E1 -13233.488,E2 -13233.488} C_VEL
LIN {X 0,Y 359.701,Z 623.6,A -85,B 0,C 180,E1 -13234.409,E2 -13234.409} C_VEL
LIN {X 0,Y 356.954,Z 621.643,A -85,B 0,C 180,E1 -13235.901,E2 -13235.901} C_VEL
LIN {X 0,Y 354.68,Z 619.715,A -85,B 0,C 180,E1 -13237.095,E2 -13237.095} C_VEL
LIN {X 0,Y 353.802,Z 617.984,A -85,B 0,C 180,E1 -13238.003,E2 -13238.003} C_VEL
LIN {X 0,Y 353.783,Z 617.323,A -85,B 0,C 180,E1 -13238.306,E2 -13238.306} C_VEL
LIN {X 0,Y 354.316,Z 612.375,A -85,B 0,C 180,E1 -13240.282,E2 -13240.282} C_VEL
LIN {X 0,Y 355.112,Z 606.028,A -85,B 0,C 180,E1 -13242.282,E2 -13242.282} C_VEL
LIN {X 0,Y 356.122,Z 599.36,A -85,B 0,C 180,E1 -13243.988,E2 -13243.988} C_VEL
LIN {X 0,Y 357.106,Z 591.503,A -85,B 0,C 180,E1 -13245.669,E2 -13245.669} C_VEL
LIN {X 0,Y 358.508,Z 581.699,A -85,B 0,C 180,E1 -13247.393,E2 -13247.393} C_VEL
LIN {X 0,Y 360.015,Z 570.979,A -85,B 0,C 180,E1 -13248.936,E2 -13248.936} C_VEL
LIN {X 0,Y 361.617,Z 559.105,A -85,B 0,C 180,E1 -13250.326,E2 -13250.326} C_VEL
LIN {X 0,Y 362.923,Z 547.433,A -85,B 0,C 180,E1 -13251.437,E2 -13251.437} C_VEL
LIN {X 0,Y 364.247,Z 533.994,A -85,B 0,C 180,E1 -13252.45,E2 -13252.45} C_VEL
LIN {X 0,Y 365.342,Z 520.34,A -85,B 0,C 180,E1 -13253.224,E2 -13253.224} C_VEL
LIN {X 0,Y 366.118,Z 506.778,A -85,B 0,C 180,E1 -13253.771,E2 -13253.771} C_VEL
LIN {X 0,Y 366.693,Z 491.671,A -85,B 0,C 180,E1 -13254.144,E2 -13254.144} C_VEL
LIN {X 0,Y 368.693,Z 398.233,A -85,B 0,C 180,E1 -13255.973,E2 -13255.973} C_VEL
LIN {X 0,Y 365.162,Z 381.256,A -85,B 0,C 180,E1 -13256.609,E2 -13256.609} C_VEL
LIN {X 0,Y 358.11,Z 364.219,A -85,B 0,C 180,E1 -13257.562,E2 -13257.562} C_VEL
LIN {X 0,Y 355.58,Z 353.107,A -85,B 0,C 180,E1 -13260.594,E2 -13260.594} C_VEL
LIN {X 0,Y 354.816,Z 349.919,A -85,B 0,C 180,E1 -13261.54,E2 -13261.54} C_VEL
LIN {X 0,Y 354.805,Z 349.918,A -85,B 0,C 180,E1 -13265.057,E2 -13265.057} C_VEL
LIN {X 0,Y 354.786,Z 349.916,A -85,B 0,C 180,E1 -13267.883,E2 -13267.883} C_VEL
LIN {X 0,Y 354.758,Z 349.92,A -85,B 0,C 180,E1 -13271.166,E2 -13271.166} C_VEL
LIN {X 0,Y 354.75,Z 349.92,A -85,B 0,C 180,E1 -13274.504,E2 -13274.504} C_VEL
LIN {X 0,Y 354.778,Z 349.916,A -85,B 0,C 180,E1 -13277.66,E2 -13277.66} C_VEL
LIN {X 0,Y 354.774,Z 349.915,A -85,B 0,C 180,E1 -13280.66,E2 -13280.66} C_VEL
LIN {X 0,Y 354.81,Z 349.912,A -85,B 0,C 180,E1 -13284.3,E2 -13284.3} C_VEL
LIN {X 0,Y 354.773,Z 349.903,A -85,B 0,C 180,E1 -13287.665,E2 -13287.665} C_VEL
LIN {X 0,Y 354.784,Z 349.911,A -85,B 0,C 180,E1 -13291.613,E2 -13291.613} C_VEL
LIN {X 0,Y 354.827,Z 349.907,A -85,B 0,C 180,E1 -13295.421,E2 -13295.421} C_VEL
LIN {X 0,Y 354.812,Z 349.901,A -85,B 0,C 180,E1 -13299.112,E2 -13299.112} C_VEL
LIN {X 0,Y 354.866,Z 349.897,A -85,B 0,C 180,E1 -13302.718,E2 -13302.718} C_VEL
LIN {X 0,Y 354.938,Z 349.895,A -85,B 0,C 180,E1 -13306.254,E2 -13306.254} C_VEL
LIN {X 0,Y 354.941,Z 349.894,A -85,B 0,C 180,E1 -13309.735,E2 -13309.735} C_VEL
LIN {X 0,Y 355.067,Z 349.88,A -85,B 0,C 180,E1 -13313.179,E2 -13313.179} C_VEL
LIN {X 0,Y 355.215,Z 349.861,A -85,B 0,C 180,E1 -13317.732,E2 -13317.732} C_VEL
LIN {X 0,Y 355.212,Z 349.864,A -85,B 0,C 180,E1 -13322.268,E2 -13322.268} C_VEL
LIN {X 0,Y 355.073,Z 349.88,A -85,B 0,C 180,E1 -13326.82,E2 -13326.82} C_VEL
LIN {X 0,Y 354.936,Z 349.897,A -85,B 0,C 180,E1 -13330.265,E2 -13330.265} C_VEL
LIN {X 0,Y 354.928,Z 349.895,A -85,B 0,C 180,E1 -13334.019,E2 -13334.019} C_VEL
LIN {X 0,Y 354.876,Z 349.903,A -85,B 0,C 180,E1 -13338.093,E2 -13338.093} C_VEL
LIN {X 0,Y 354.792,Z 349.897,A -85,B 0,C 180,E1 -13342.109,E2 -13342.109} C_VEL
LIN {X 0,Y 354.786,Z 349.915,A -85,B 0,C 180,E1 -13345.836,E2 -13345.836} C_VEL
LIN {X 0,Y 354.78,Z 349.903,A -85,B 0,C 180,E1 -13349.685,E2 -13349.685} C_VEL
LIN {X 0,Y 354.772,Z 349.919,A -85,B 0,C 180,E1 -13352.335,E2 -13352.335} C_VEL
LIN {X 0,Y 354.806,Z 349.913,A -85,B 0,C 180,E1 -13355.699,E2 -13355.699} C_VEL
LIN {X 0,Y 354.757,Z 349.918,A -85,B 0,C 180,E1 -13359.414,E2 -13359.414} C_VEL
LIN {X 0,Y 354.77,Z 349.917,A -85,B 0,C 180,E1 -13362.867,E2 -13362.867} C_VEL
LIN {X 0,Y 354.752,Z 349.922,A -85,B 0,C 180,E1 -13366.104,E2 -13366.104} C_VEL
LIN {X 0,Y 354.753,Z 349.922,A -85,B 0,C 180,E1 -13369.177,E2 -13369.177} C_VEL
LIN {X 0,Y 354.789,Z 349.92,A -85,B 0,C 180,E1 -13372.406,E2 -13372.406} C_VEL
LIN {X 0,Y 354.8,Z 349.917,A -85,B 0,C 180,E1 -13374.942,E2 -13374.942} C_VEL
LIN {X 0,Y 354.829,Z 350.018,A -85,B 0,C 180,E1 -13377.295,E2 -13377.295} C_VEL
LIN {X 0,Y 357.757,Z 362.264,A -85,B 0,C 180,E1 -13380.588,E2 -13380.588} C_VEL
LIN {X 0,Y 359.464,Z 370.142,A -85,B 0,C 180,E1 -13382.602,E2 -13382.602} C_VEL
LIN {X 0,Y 363.374,Z 380.217,A -85,B 0,C 180,E1 -13383.139,E2 -13383.139} C_VEL
LIN {X 0,Y 368.077,Z 403.957,A -85,B 0,C 180,E1 -13384.014,E2 -13384.014} C_VEL
LIN {X 0,Y 368.565,Z 408.412,A -85,B 0,C 180,E1 -13384.145,E2 -13384.145} C_VEL
LIN {X 0,Y 366.348,Z 507.156,A -85,B 0,C 180,E1 -13386.095,E2 -13386.095} C_VEL
LIN {X 0,Y 365.496,Z 521.978,A -85,B 0,C 180,E1 -13386.599,E2 -13386.599} C_VEL
LIN {X 0,Y 364.4,Z 536.022,A -85,B 0,C 180,E1 -13387.313,E2 -13387.313} C_VEL
LIN {X 0,Y 363.242,Z 548.534,A -85,B 0,C 180,E1 -13388.165,E2 -13388.165} C_VEL
LIN {X 0,Y 361.872,Z 561.205,A -85,B 0,C 180,E1 -13389.267,E2 -13389.267} C_VEL
LIN {X 0,Y 360.43,Z 572.598,A -85,B 0,C 180,E1 -13390.495,E2 -13390.495} C_VEL
LIN {X 0,Y 358.751,Z 584.23,A -85,B 0,C 180,E1 -13392.03,E2 -13392.03} C_VEL
LIN {X 0,Y 357.269,Z 594.634,A -85,B 0,C 180,E1 -13393.723,E2 -13393.723} C_VEL
LIN {X 0,Y 356.165,Z 603.055,A -85,B 0,C 180,E1 -13395.395,E2 -13395.395} C_VEL
LIN {X 0,Y 355.095,Z 611.436,A -85,B 0,C 180,E1 -13397.427,E2 -13397.427} C_VEL
LIN {X 0,Y 354.302,Z 617.188,A -85,B 0,C 180,E1 -13399.14,E2 -13399.14} C_VEL
LIN {X 0,Y 353.824,Z 621.901,A -85,B 0,C 180,E1 -13400.859,E2 -13400.859} C_VEL
LIN {X 0,Y 353.415,Z 626.79,A -85,B 0,C 180,E1 -13403.149,E2 -13403.149} C_VEL
LIN {X 0,Y 353.255,Z 630.186,A -85,B 0,C 180,E1 -13405.437,E2 -13405.437} C_VEL
LIN {X 0,Y 353.131,Z 632.19,A -85,B 0,C 180,E1 -13407.721,E2 -13407.721} C_VEL
LIN {X 0,Y 353.173,Z 632.851,A -85,B 0,C 180,E1 -13410.002,E2 -13410.002} C_VEL
LIN {X 0,Y 353.131,Z 632.178,A -85,B 0,C 180,E1 -13412.283,E2 -13412.283} C_VEL
LIN {X 0,Y 353.257,Z 630.162,A -85,B 0,C 180,E1 -13414.566,E2 -13414.566} C_VEL
LIN {X 0,Y 353.428,Z 626.758,A -85,B 0,C 180,E1 -13416.854,E2 -13416.854} C_VEL
LIN {X 0,Y 353.827,Z 621.864,A -85,B 0,C 180,E1 -13419.145,E2 -13419.145} C_VEL
LIN {X 0,Y 354.305,Z 617.139,A -85,B 0,C 180,E1 -13420.863,E2 -13420.863} C_VEL
LIN {X 0,Y 355.255,Z 610.288,A -85,B 0,C 180,E1 -13422.861,E2 -13422.861} C_VEL
LIN {X 0,Y 356.254,Z 601.785,A -85,B 0,C 180,E1 -13424.862,E2 -13424.862} C_VEL
LIN {X 0,Y 357.525,Z 592.911,A -85,B 0,C 180,E1 -13426.562,E2 -13426.562} C_VEL
LIN {X 0,Y 359.066,Z 582.165,A -85,B 0,C 180,E1 -13428.252,E2 -13428.252} C_VEL
LIN {X 0,Y 360.565,Z 571.285,A -85,B 0,C 180,E1 -13429.649,E2 -13429.649} C_VEL
LIN {X 0,Y 362.005,Z 559.635,A -85,B 0,C 180,E1 -13430.874,E2 -13430.874} C_VEL
LIN {X 0,Y 363.421,Z 546.732,A -85,B 0,C 180,E1 -13431.961,E2 -13431.961} C_VEL
LIN {X 0,Y 364.59,Z 533.476,A -85,B 0,C 180,E1 -13432.828,E2 -13432.828} C_VEL
LIN {X 0,Y 365.64,Z 519.998,A -85,B 0,C 180,E1 -13433.47,E2 -13433.47} C_VEL
LIN {X 0,Y 366.303,Z 506.456,A -85,B 0,C 180,E1 -13433.912,E2 -13433.912} C_VEL
LIN {X 0,Y 367.932,Z 436.387,A -85,B 0,C 180,E1 -13435.294,E2 -13435.294} C_VEL
LIN {X 0,Y 368.436,Z 406.112,A -85,B 0,C 180,E1 -13435.898,E2 -13435.898} C_VEL
LIN {X 0,Y 364.162,Z 383.726,A -85,B 0,C 180,E1 -13436.732,E2 -13436.732} C_VEL
LIN {X 0,Y 364.022,Z 379.453,A -85,B 0,C 180,E1 -13437.154,E2 -13437.154} C_VEL
LIN {X 0,Y 361.912,Z 372.82,A -85,B 0,C 180,E1 -13438.191,E2 -13438.191} C_VEL
LIN {X 0,Y 359.837,Z 365.793,A -85,B 0,C 180,E1 -13439.397,E2 -13439.397} C_VEL
LIN {X 0,Y 356.643,Z 356.021,A -85,B 0,C 180,E1 -13441.479,E2 -13441.479} C_VEL
LIN {X 0,Y 354.835,Z 349.908,A -85,B 0,C 180,E1 -13443.068,E2 -13443.068} C_VEL
LIN {X 0,Y 354.802,Z 349.91,A -85,B 0,C 180,E1 -13446.461,E2 -13446.461} C_VEL
LIN {X 0,Y 354.829,Z 349.911,A -85,B 0,C 180,E1 -13449.425,E2 -13449.425} C_VEL
LIN {X 0,Y 354.794,Z 349.914,A -85,B 0,C 180,E1 -13452.868,E2 -13452.868} C_VEL
LIN {X 0,Y 354.772,Z 349.915,A -85,B 0,C 180,E1 -13456.104,E2 -13456.104} C_VEL
LIN {X 0,Y 354.794,Z 349.917,A -85,B 0,C 180,E1 -13459.18,E2 -13459.18} C_VEL
LIN {X 0,Y 354.813,Z 349.912,A -85,B 0,C 180,E1 -13462.403,E2 -13462.403} C_VEL
LIN {X 0,Y 354.836,Z 349.971,A -85,B 0,C 180,E1 -13464.026,E2 -13464.026} C_VEL
LIN {X 0,Y 358.369,Z 358.734,A -85,B 0,C 180,E1 -13467.49,E2 -13467.49} C_VEL
LIN {X 0,Y 361.054,Z 366.178,A -85,B 0,C 180,E1 -13469.951,E2 -13469.951} C_VEL
LIN {X 0,Y 363.654,Z 375.978,A -85,B 0,C 180,E1 -13472.75,E2 -13472.75} C_VEL
LIN {X 0,Y 364.763,Z 382.038,A -85,B 0,C 180,E1 -13474.31,E2 -13474.31} C_VEL
LIN {X 0,Y 364.951,Z 384.541,A -85,B 0,C 180,E1 -13474.839,E2 -13474.839} C_VEL
LIN {X 0,Y 368.367,Z 397.295,A -85,B 0,C 180,E1 -13475.842,E2 -13475.842} C_VEL
LIN {X 0,Y 370.499,Z 407.651,A -85,B 0,C 180,E1 -13476.525,E2 -13476.525} C_VEL
LIN {X 0,Y 365.965,Z 484.578,A -85,B 0,C 180,E1 -13478.895,E2 -13478.895} C_VEL
LIN {X 0,Y 365.12,Z 499.475,A -85,B 0,C 180,E1 -13479.434,E2 -13479.434} C_VEL
LIN {X 0,Y 364.183,Z 512.199,A -85,B 0,C 180,E1 -13480.115,E2 -13480.115} C_VEL
LIN {X 0,Y 363.143,Z 523.752,A -85,B 0,C 180,E1 -13480.938,E2 -13480.938} C_VEL
LIN {X 0,Y 361.837,Z 535.764,A -85,B 0,C 180,E1 -13482.028,E2 -13482.028} C_VEL
LIN {X 0,Y 360.585,Z 545.695,A -85,B 0,C 180,E1 -13483.151,E2 -13483.151} C_VEL
LIN {X 0,Y 359.356,Z 554.774,A -85,B 0,C 180,E1 -13484.401,E2 -13484.401} C_VEL
LIN {X 0,Y 358.124,Z 563.201,A -85,B 0,C 180,E1 -13485.8,E2 -13485.8} C_VEL
LIN {X 0,Y 356.856,Z 571.407,A -85,B 0,C 180,E1 -13487.489,E2 -13487.489} C_VEL
LIN {X 0,Y 355.901,Z 577.994,A -85,B 0,C 180,E1 -13489.187,E2 -13489.187} C_VEL
LIN {X 0,Y 355.065,Z 583.236,A -85,B 0,C 180,E1 -13490.889,E2 -13490.889} C_VEL
LIN {X 0,Y 354.568,Z 586.72,A -85,B 0,C 180,E1 -13492.343,E2 -13492.343} C_VEL
LIN {X 0,Y 353.886,Z 590.208,A -85,B 0,C 180,E1 -13494.301,E2 -13494.301} C_VEL
LIN {X 0,Y 353.802,Z 591.567,A -85,B 0,C 180,E1 -13495.443,E2 -13495.443} C_VEL
LIN {X 0,Y 353.723,Z 592.491,A -85,B 0,C 180,E1 -13496.583,E2 -13496.583} C_VEL
LIN {X 0,Y 353.572,Z 593.015,A -85,B 0,C 180,E1 -13497.722,E2 -13497.722} C_VEL
LIN {X 0,Y 353.448,Z 593.085,A -85,B 0,C 180,E1 -13498.861,E2 -13498.861} C_VEL
LIN {X 0,Y 353.383,Z 592.701,A -85,B 0,C 180,E1 -13500,E2 -13500} C_VEL
LIN {X 0,Y 353.36,Z 591.904,A -85,B 0,C 180,E1 -13501.14,E2 -13501.14} C_VEL
LIN {X 0,Y 353.365,Z 590.66,A -85,B 0,C 180,E1 -13502.28,E2 -13502.28} C_VEL
LIN {X 0,Y 353.45,Z 587.927,A -85,B 0,C 180,E1 -13503.991,E2 -13503.991} C_VEL
LIN {X 0,Y 353.596,Z 584.099,A -85,B 0,C 180,E1 -13505.704,E2 -13505.704} C_VEL
LIN {X 0,Y 353.849,Z 579.074,A -85,B 0,C 180,E1 -13507.418,E2 -13507.418} C_VEL
LIN {X 0,Y 354.217,Z 572.709,A -85,B 0,C 180,E1 -13509.133,E2 -13509.133} C_VEL
LIN {X 0,Y 354.771,Z 564.752,A -85,B 0,C 180,E1 -13510.848,E2 -13510.848} C_VEL
LIN {X 0,Y 355.464,Z 554.786,A -85,B 0,C 180,E1 -13512.561,E2 -13512.561} C_VEL
LIN {X 0,Y 356.2,Z 544.443,A -85,B 0,C 180,E1 -13513.987,E2 -13513.987} C_VEL
LIN {X 0,Y 356.882,Z 533.487,A -85,B 0,C 180,E1 -13515.211,E2 -13515.211} C_VEL
LIN {X 0,Y 357.552,Z 521.612,A -85,B 0,C 180,E1 -13516.266,E2 -13516.266} C_VEL
LIN {X 0,Y 358.336,Z 508.11,A -85,B 0,C 180,E1 -13517.183,E2 -13517.183} C_VEL
LIN {X 0,Y 358.821,Z 494.194,A -85,B 0,C 180,E1 -13517.858,E2 -13517.858} C_VEL
LIN {X 0,Y 359.25,Z 479.471,A -85,B 0,C 180,E1 -13518.315,E2 -13518.315} C_VEL
LIN {X 0,Y 361.177,Z 402.537,A -85,B 0,C 180,E1 -13520.335,E2 -13520.335} C_VEL
LIN {X 0,Y 357.731,Z 379.398,A -85,B 0,C 180,E1 -13521.124,E2 -13521.124} C_VEL
LIN {X 0,Y 358.247,Z 367.733,A -85,B 0,C 180,E1 -13523.407,E2 -13523.407} C_VEL
LIN {X 0,Y 356.255,Z 356.66,A -85,B 0,C 180,E1 -13525.722,E2 -13525.722} C_VEL
LIN {X 0,Y 354.9,Z 349.903,A -85,B 0,C 180,E1 -13527.175,E2 -13527.175} C_VEL
LIN {X 0,Y 354.861,Z 349.908,A -85,B 0,C 180,E1 -13529.678,E2 -13529.678} C_VEL
LIN {X 0,Y 354.813,Z 349.912,A -85,B 0,C 180,E1 -13533.701,E2 -13533.701} C_VEL
LIN {X 0,Y 354.802,Z 349.914,A -85,B 0,C 180,E1 -13536.459,E2 -13536.459} C_VEL
LIN {X 0,Y 354.774,Z 349.917,A -85,B 0,C 180,E1 -13539.412,E2 -13539.412} C_VEL
LIN {X 0,Y 354.791,Z 349.914,A -85,B 0,C 180,E1 -13542.866,E2 -13542.866} C_VEL
LIN {X 0,Y 354.772,Z 349.92,A -85,B 0,C 180,E1 -13546.103,E2 -13546.103} C_VEL
LIN {X 0,Y 354.771,Z 349.919,A -85,B 0,C 180,E1 -13549.175,E2 -13549.175} C_VEL
LIN {X 0,Y 354.804,Z 349.914,A -85,B 0,C 180,E1 -13552.404,E2 -13552.404} C_VEL
LIN {X 0,Y 354.813,Z 349.91,A -85,B 0,C 180,E1 -13554.939,E2 -13554.939} C_VEL
LIN {X 0,Y 354.809,Z 349.931,A -85,B 0,C 180,E1 -13558.617,E2 -13558.617} C_VEL
LIN {X 0,Y 357.295,Z 360.338,A -85,B 0,C 180,E1 -13561.509,E2 -13561.509} C_VEL
LIN {X 0,Y 358.102,Z 364.247,A -85,B 0,C 180,E1 -13562.552,E2 -13562.552} C_VEL
LIN {X 0,Y 365.551,Z 382.337,A -85,B 0,C 180,E1 -13563.551,E2 -13563.551} C_VEL
LIN {X 0,Y 368.695,Z 398.787,A -85,B 0,C 180,E1 -13564.145,E2 -13564.145} C_VEL
LIN {X 0,Y 366.449,Z 499.809,A -85,B 0,C 180,E1 -13566.136,E2 -13566.136} C_VEL
LIN {X 0,Y 365.731,Z 514.333,A -85,B 0,C 180,E1 -13566.612,E2 -13566.612} C_VEL
LIN {X 0,Y 364.731,Z 527.579,A -85,B 0,C 180,E1 -13567.256,E2 -13567.256} C_VEL
LIN {X 0,Y 363.572,Z 540.694,A -85,B 0,C 180,E1 -13568.123,E2 -13568.123} C_VEL
LIN {X 0,Y 362.37,Z 552.528,A -85,B 0,C 180,E1 -13569.121,E2 -13569.121} C_VEL
LIN {X 0,Y 360.925,Z 564.491,A -85,B 0,C 180,E1 -13570.371,E2 -13570.371} C_VEL
LIN {X 0,Y 359.368,Z 575.403,A -85,B 0,C 180,E1 -13571.764,E2 -13571.764} C_VEL
LIN {X 0,Y 358.069,Z 584.542,A -85,B 0,C 180,E1 -13573.17,E2 -13573.17} C_VEL
LIN {X 0,Y 356.841,Z 593.41,A -85,B 0,C 180,E1 -13574.809,E2 -13574.809} C_VEL
LIN {X 0,Y 355.83,Z 601.324,A -85,B 0,C 180,E1 -13576.579,E2 -13576.579} C_VEL
LIN {X 0,Y 354.749,Z 608.599,A -85,B 0,C 180,E1 -13578.572,E2 -13578.572} C_VEL
LIN {X 0,Y 354.174,Z 613.689,A -85,B 0,C 180,E1 -13580.288,E2 -13580.288} C_VEL
LIN {X 0,Y 353.636,Z 618.964,A -85,B 0,C 180,E1 -13582.576,E2 -13582.576} C_VEL
LIN {X 0,Y 353.427,Z 621.906,A -85,B 0,C 180,E1 -13584.292,E2 -13584.292} C_VEL
LIN {X 0,Y 353.234,Z 624.614,A -85,B 0,C 180,E1 -13586.576,E2 -13586.576} C_VEL
LIN {X 0,Y 353.157,Z 625.974,A -85,B 0,C 180,E1 -13588.858,E2 -13588.858} C_VEL
LIN {X 0,Y 353.157,Z 626.009,A -85,B 0,C 180,E1 -13591.139,E2 -13591.139} C_VEL
LIN {X 0,Y 353.235,Z 624.643,A -85,B 0,C 180,E1 -13593.497,E2 -13593.497} C_VEL
LIN {X 0,Y 353.399,Z 622.075,A -85,B 0,C 180,E1 -13595.705,E2 -13595.705} C_VEL
LIN {X 0,Y 353.721,Z 618.001,A -85,B 0,C 180,E1 -13597.993,E2 -13597.993} C_VEL
LIN {X 0,Y 353.783,Z 617.323,A -85,B 0,C 180,E1 -13598.306,E2 -13598.306} C_VEL
LIN {X 0,Y 353.334,Z 615.315,A -85,B 0,C 180,E1 -13599.204,E2 -13599.204} C_VEL
LIN {X 0,Y 350.915,Z 611.724,A -85,B 0,C 180,E1 -13600.656,E2 -13600.656} C_VEL
LIN {X 0,Y 348.643,Z 607.568,A -85,B 0,C 180,E1 -13602.086,E2 -13602.086} C_VEL
LIN {X 0,Y 348.426,Z 604.675,A -85,B 0,C 180,E1 -13602.933,E2 -13602.933} C_VEL
LIN {X 0,Y 349.447,Z 596.978,A -85,B 0,C 180,E1 -13604.851,E2 -13604.851} C_VEL
LIN {X 0,Y 350.711,Z 588.442,A -85,B 0,C 180,E1 -13606.59,E2 -13606.59} C_VEL
LIN {X 0,Y 352.248,Z 578.123,A -85,B 0,C 180,E1 -13608.313,E2 -13608.313} C_VEL
LIN {X 0,Y 353.961,Z 566.578,A -85,B 0,C 180,E1 -13609.876,E2 -13609.876} C_VEL
LIN {X 0,Y 355.485,Z 555.087,A -85,B 0,C 180,E1 -13611.144,E2 -13611.144} C_VEL
LIN {X 0,Y 356.902,Z 542.181,A -85,B 0,C 180,E1 -13612.291,E2 -13612.291} C_VEL
LIN {X 0,Y 358.098,Z 529.259,A -85,B 0,C 180,E1 -13613.186,E2 -13613.186} C_VEL
LIN {X 0,Y 359.175,Z 515.069,A -85,B 0,C 180,E1 -13613.914,E2 -13613.914} C_VEL
LIN {X 0,Y 359.961,Z 501.115,A -85,B 0,C 180,E1 -13614.395,E2 -13614.395} C_VEL
LIN {X 0,Y 362.281,Z 405.852,A -85,B 0,C 180,E1 -13616.303,E2 -13616.303} C_VEL
LIN {X 0,Y 362.284,Z 399.133,A -85,B 0,C 180,E1 -13616.449,E2 -13616.449} C_VEL
LIN {X 0,Y 358.999,Z 383.494,A -85,B 0,C 180,E1 -13617.054,E2 -13617.054} C_VEL
LIN {X 0,Y 350.936,Z 364.311,A -85,B 0,C 180,E1 -13618.17,E2 -13618.17} C_VEL
LIN {X 0,Y 348.321,Z 353.19,A -85,B 0,C 180,E1 -13621.3,E2 -13621.3} C_VEL
LIN {X 0,Y 347.74,Z 350.799,A -85,B 0,C 180,E1 -13622.035,E2 -13622.035} C_VEL
LIN {X 0,Y 347.781,Z 350.791,A -85,B 0,C 180,E1 -13625.874,E2 -13625.874} C_VEL
LIN {X 0,Y 347.723,Z 350.797,A -85,B 0,C 180,E1 -13628.794,E2 -13628.794} C_VEL
LIN {X 0,Y 347.731,Z 350.794,A -85,B 0,C 180,E1 -13631.83,E2 -13631.83} C_VEL
LIN {X 0,Y 347.693,Z 350.8,A -85,B 0,C 180,E1 -13635.026,E2 -13635.026} C_VEL
LIN {X 0,Y 347.731,Z 350.795,A -85,B 0,C 180,E1 -13638.397,E2 -13638.397} C_VEL
LIN {X 0,Y 347.745,Z 350.783,A -85,B 0,C 180,E1 -13642.677,E2 -13642.677} C_VEL
LIN {X 0,Y 347.737,Z 350.79,A -85,B 0,C 180,E1 -13645.955,E2 -13645.955} C_VEL
LIN {X 0,Y 347.723,Z 350.794,A -85,B 0,C 180,E1 -13649.649,E2 -13649.649} C_VEL
LIN {X 0,Y 347.725,Z 350.774,A -85,B 0,C 180,E1 -13653.599,E2 -13653.599} C_VEL
LIN {X 0,Y 347.743,Z 350.79,A -85,B 0,C 180,E1 -13656.158,E2 -13656.158} C_VEL
LIN {X 0,Y 347.784,Z 350.771,A -85,B 0,C 180,E1 -13659.907,E2 -13659.907} C_VEL
LIN {X 0,Y 347.817,Z 350.781,A -85,B 0,C 180,E1 -13663.567,E2 -13663.567} C_VEL
LIN {X 0,Y 347.875,Z 350.774,A -85,B 0,C 180,E1 -13667.16,E2 -13667.16} C_VEL
LIN {X 0,Y 347.92,Z 350.767,A -85,B 0,C 180,E1 -13670.7,E2 -13670.7} C_VEL
LIN {X 0,Y 348.02,Z 350.759,A -85,B 0,C 180,E1 -13674.205,E2 -13674.205} C_VEL
LIN {X 0,Y 348.177,Z 350.738,A -85,B 0,C 180,E1 -13677.686,E2 -13677.686} C_VEL
LIN {X 0,Y 348.128,Z 350.744,A -85,B 0,C 180,E1 -13681.157,E2 -13681.157} C_VEL
LIN {X 0,Y 348.174,Z 350.741,A -85,B 0,C 180,E1 -13682.314,E2 -13682.314} C_VEL
LIN {X 0,Y 348.04,Z 350.755,A -85,B 0,C 180,E1 -13686.959,E2 -13686.959} C_VEL
LIN {X 0,Y 347.876,Z 350.779,A -85,B 0,C 180,E1 -13690.476,E2 -13690.476} C_VEL
LIN {X 0,Y 347.885,Z 350.773,A -85,B 0,C 180,E1 -13694.15,E2 -13694.15} C_VEL
LIN {X 0,Y 347.815,Z 350.784,A -85,B 0,C 180,E1 -13698.26,E2 -13698.26} C_VEL
LIN {X 0,Y 347.75,Z 350.776,A -85,B 0,C 180,E1 -13701.625,E2 -13701.625} C_VEL
LIN {X 0,Y 347.723,Z 350.794,A -85,B 0,C 180,E1 -13705.115,E2 -13705.115} C_VEL
LIN {X 0,Y 347.716,Z 350.79,A -85,B 0,C 180,E1 -13707.702,E2 -13707.702} C_VEL
LIN {X 0,Y 347.723,Z 350.788,A -85,B 0,C 180,E1 -13710.35,E2 -13710.35} C_VEL
LIN {X 0,Y 347.736,Z 350.792,A -85,B 0,C 180,E1 -13714.045,E2 -13714.045} C_VEL
LIN {X 0,Y 347.742,Z 350.793,A -85,B 0,C 180,E1 -13717.323,E2 -13717.323} C_VEL
LIN {X 0,Y 347.684,Z 350.803,A -85,B 0,C 180,E1 -13720.304,E2 -13720.304} C_VEL
LIN {X 0,Y 347.71,Z 350.796,A -85,B 0,C 180,E1 -13723.41,E2 -13723.41} C_VEL
LIN {X 0,Y 347.712,Z 350.8,A -85,B 0,C 180,E1 -13726.689,E2 -13726.689} C_VEL
LIN {X 0,Y 347.691,Z 350.804,A -85,B 0,C 180,E1 -13730.184,E2 -13730.184} C_VEL
LIN {X 0,Y 347.745,Z 350.796,A -85,B 0,C 180,E1 -13732.68,E2 -13732.68} C_VEL
LIN {X 0,Y 347.74,Z 350.796,A -85,B 0,C 180,E1 -13735.958,E2 -13735.958} C_VEL
LIN {X 0,Y 347.769,Z 350.828,A -85,B 0,C 180,E1 -13736.772,E2 -13736.772} C_VEL
LIN {X 0,Y 350.516,Z 362.194,A -85,B 0,C 180,E1 -13739.919,E2 -13739.919} C_VEL
LIN {X 0,Y 352.274,Z 370.142,A -85,B 0,C 180,E1 -13741.995,E2 -13741.995} C_VEL
